REGION Network 6: CY75 interface K-reserveTakeStopperCylinder3_1
   RUNG wire#powerrail
      Contact( #AlwaysON )
      wire#w1
      Contact( #E_stop )
      wire#w2
      Coil( "ST10Cylinder".Cy[75].In.GoWorkInterlock )
   END_RUNG
   RUNG wire#w2
      Coil( "ST10Cylinder".Cy[75].In.GoHomeInterlock )
   END_RUNG
   RUNG wire#w1
      I_Contact( #AlwaysON )
      Coil( "ST10Cylinder".Cy[75].In.Error )
   END_RUNG
   // the same network as SCL:
   "ST10Cylinder".Cy[75].In.GoWorkInterlock := #AlwaysON AND #E_stop;
   "ST10Cylinder".Cy[75].In.GoHomeInterlock := #AlwaysON AND #E_stop;
   "ST10Cylinder".Cy[75].In.Error := #AlwaysON AND NOT #AlwaysON;
END_REGION

REGION Network 7: CY76 interface K-reserveTakeStopperCylinder3_2
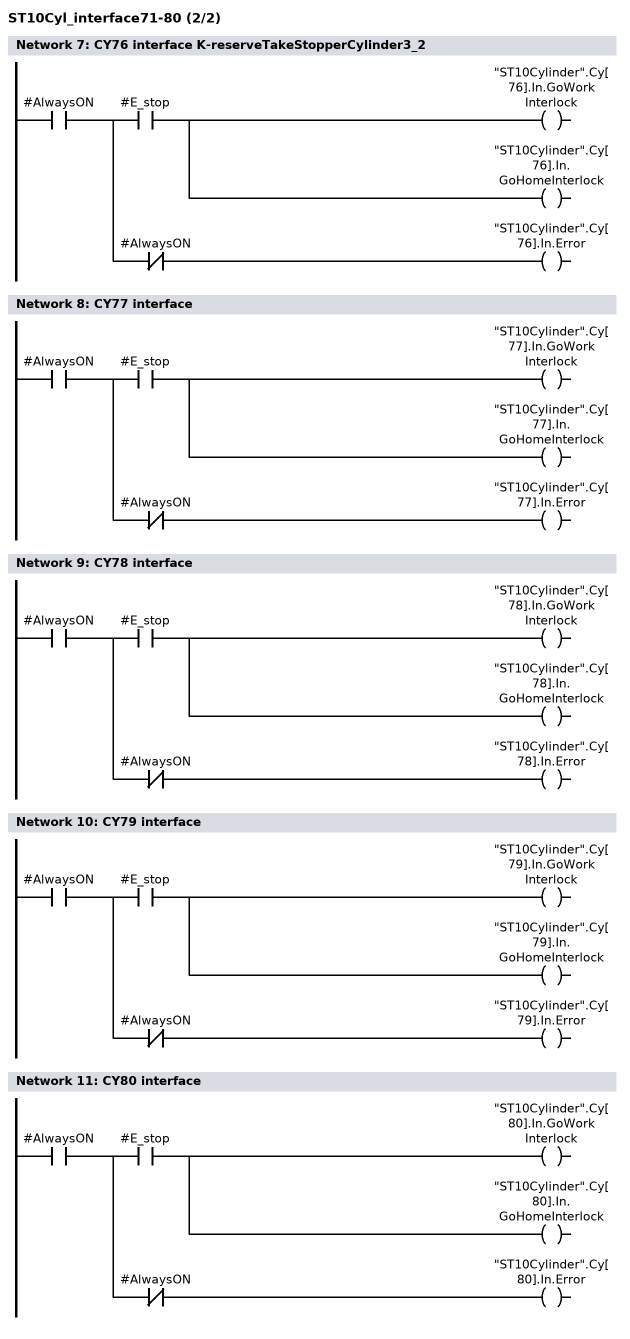
   RUNG wire#powerrail
      Contact( #AlwaysON )
      wire#w1
      Contact( #E_stop )
      wire#w2
      Coil( "ST10Cylinder".Cy[76].In.GoWorkInterlock )
   END_RUNG
   RUNG wire#w2
      Coil( "ST10Cylinder".Cy[76].In.GoHomeInterlock )
   END_RUNG
   RUNG wire#w1
      I_Contact( #AlwaysON )
      Coil( "ST10Cylinder".Cy[76].In.Error )
   END_RUNG
   // the same network as SCL:
   "ST10Cylinder".Cy[76].In.GoWorkInterlock := #AlwaysON AND #E_stop;
   "ST10Cylinder".Cy[76].In.GoHomeInterlock := #AlwaysON AND #E_stop;
   "ST10Cylinder".Cy[76].In.Error := #AlwaysON AND NOT #AlwaysON;
END_REGION

REGION Network 8: CY77 interface
   RUNG wire#powerrail
      Contact( #AlwaysON )
      wire#w1
      Contact( #E_stop )
      wire#w2
      Coil( "ST10Cylinder".Cy[77].In.GoWorkInterlock )
   END_RUNG
   RUNG wire#w2
      Coil( "ST10Cylinder".Cy[77].In.GoHomeInterlock )
   END_RUNG
   RUNG wire#w1
      I_Contact( #AlwaysON )
      Coil( "ST10Cylinder".Cy[77].In.Error )
   END_RUNG
   // the same network as SCL:
   "ST10Cylinder".Cy[77].In.GoWorkInterlock := #AlwaysON AND #E_stop;
   "ST10Cylinder".Cy[77].In.GoHomeInterlock := #AlwaysON AND #E_stop;
   "ST10Cylinder".Cy[77].In.Error := #AlwaysON AND NOT #AlwaysON;
END_REGION

REGION Network 9: CY78 interface
   RUNG wire#powerrail
      Contact( #AlwaysON )
      wire#w1
      Contact( #E_stop )
      wire#w2
      Coil( "ST10Cylinder".Cy[78].In.GoWorkInterlock )
   END_RUNG
   RUNG wire#w2
      Coil( "ST10Cylinder".Cy[78].In.GoHomeInterlock )
   END_RUNG
   RUNG wire#w1
      I_Contact( #AlwaysON )
      Coil( "ST10Cylinder".Cy[78].In.Error )
   END_RUNG
   // the same network as SCL:
   "ST10Cylinder".Cy[78].In.GoWorkInterlock := #AlwaysON AND #E_stop;
   "ST10Cylinder".Cy[78].In.GoHomeInterlock := #AlwaysON AND #E_stop;
   "ST10Cylinder".Cy[78].In.Error := #AlwaysON AND NOT #AlwaysON;
END_REGION

REGION Network 10: CY79 interface
   RUNG wire#powerrail
      Contact( #AlwaysON )
      wire#w1
      Contact( #E_stop )
      wire#w2
      Coil( "ST10Cylinder".Cy[79].In.GoWorkInterlock )
   END_RUNG
   RUNG wire#w2
      Coil( "ST10Cylinder".Cy[79].In.GoHomeInterlock )
   END_RUNG
   RUNG wire#w1
      I_Contact( #AlwaysON )
      Coil( "ST10Cylinder".Cy[79].In.Error )
   END_RUNG
   // the same network as SCL:
   "ST10Cylinder".Cy[79].In.GoWorkInterlock := #AlwaysON AND #E_stop;
   "ST10Cylinder".Cy[79].In.GoHomeInterlock := #AlwaysON AND #E_stop;
   "ST10Cylinder".Cy[79].In.Error := #AlwaysON AND NOT #AlwaysON;
END_REGION

REGION Network 11: CY80 interface
   RUNG wire#powerrail
      Contact( #AlwaysON )
      wire#w1
      Contact( #E_stop )
      wire#w2
      Coil( "ST10Cylinder".Cy[80].In.GoWorkInterlock )
   END_RUNG
   RUNG wire#w2
      Coil( "ST10Cylinder".Cy[80].In.GoHomeInterlock )
   END_RUNG
   RUNG wire#w1
      I_Contact( #AlwaysON )
      Coil( "ST10Cylinder".Cy[80].In.Error )
   END_RUNG
   // the same network as SCL:
   "ST10Cylinder".Cy[80].In.GoWorkInterlock := #AlwaysON AND #E_stop;
   "ST10Cylinder".Cy[80].In.GoHomeInterlock := #AlwaysON AND #E_stop;
   "ST10Cylinder".Cy[80].In.Error := #AlwaysON AND NOT #AlwaysON;
END_REGION
END_FUNCTION

FUNCTION "ST10Cyl_interface81-90" : Void   // FC1028, LAD
{ S7_Optimized_Access := 'FALSE' }
// stored: AutoNumber false, SetENOAutomatically false
   VAR_INPUT
      AlwaysON : Bool;
      E_stop : Bool;
   END_VAR
   VAR_TEMP
      tTest : Bool;
   END_VAR
BEGIN

REGION Network 1 (SCL): Cylinder 81-90 IO Interface (SCL)
   (*
   //Cylinder81 IO  L-UnloadingTransCylinder
   //Input
   "ST10Cylinder".Cy[81].In.WorkPositionSensor := "iL-UnloadingTransCylinderInWP";
   "ST10Cylinder".Cy[81].In.HomePositionSensor := "iL-UnloadingTransCylinderInHP";
   //Output
   "oL-UnloadingTransCylinderToWP" := "ST10Cylinder".Cy[81].Out.GoWorkPosition;
   "oL-UnloadingTransCylinderToHP" := "ST10Cylinder".Cy[81].Out.GoHomePosition;

   //Cylinder82 IO  L-UnloadingTransPalletLocationCylinder
   //Input
   "ST10Cylinder".Cy[82].In.WorkPositionSensor := "iL-UnloadingTransPalletLocationCylinderInWP";
   "ST10Cylinder".Cy[82].In.HomePositionSensor := "iL-UnloadingTransPalletLocationCylinderInHP";
   //Output
   "oL-UnloadingTransPalletLocationCylinderToWP" := "ST10Cylinder".Cy[82].Out.GoWorkPosition;
   "oL-UnloadingTransPalletLocationCylinderToHP" := "ST10Cylinder".Cy[82].Out.GoHomePosition;

   //Cylinder83 IO  L-UnloadingStopperCylinder1_1
   //Input
   "ST10Cylinder".Cy[83].In.WorkPositionSensor := "oL-UnloadingStopperCylinder1_1";
   "ST10Cylinder".Cy[83].In.HomePositionSensor := NOT "oL-UnloadingStopperCylinder1_1";
   //Output
   "oL-UnloadingStopperCylinder1_1" := "ST10Cylinder".Cy[83].Out.GoWorkPosition;
   //"oI-0030TrayLoading8trayStopperCylinderToHP" := "ST10Cylinder".Cy[83].Out.GoHomePosition;

   //Cylinder84 IO  L-UnloadingStopperCylinder1_2
   //Input
   "ST10Cylinder".Cy[84].In.WorkPositionSensor := "oL-UnloadingStopperCylinder1_2";
   "ST10Cylinder".Cy[84].In.HomePositionSensor := NOT "oL-UnloadingStopperCylinder1_2";
   //Output
   "oL-UnloadingStopperCylinder1_2" := "ST10Cylinder".Cy[84].Out.GoWorkPosition;
   //"oI-0080TrayLoadingTaketrayCylinderToHP" := "ST10Cylinder".Cy[84].Out.GoHomePosition;

   //Cylinder85 IO  L-UnloadingStopperCylinder2_1
   //Input
   "ST10Cylinder".Cy[85].In.WorkPositionSensor := "oL-UnloadingStopperCylinder2_1";
   "ST10Cylinder".Cy[85].In.HomePositionSensor := NOT "oL-UnloadingStopperCylinder2_1";
   //Output
   "oL-UnloadingStopperCylinder2_1" := "ST10Cylinder".Cy[85].Out.GoWorkPosition;
   //"oI-0050TrayLoadingTrayCylinderToHP" := "ST10Cylinder".Cy[85].Out.GoHomePosition;

   //Cylinder86  L-UnloadingStopperCylinder2_2
   //Input
   "ST10Cylinder".Cy[86].In.WorkPositionSensor := "oL-UnloadingStopperCylinder2_2";
   "ST10Cylinder".Cy[86].In.HomePositionSensor := NOT "oL-UnloadingStopperCylinder2_2";
   //Output
   "oL-UnloadingStopperCylinder2_2" := "ST10Cylinder".Cy[86].Out.GoWorkPosition;
   //"oI-0080TrayLoadingTraySupportCylinder1ToHP" := "ST10Cylinder".Cy[86].Out.GoHomePosition;

   //Cylinder87 L-UnloadingStopperCylinder3_1
   //Input
   "ST10Cylinder".Cy[87].In.WorkPositionSensor := "oL-UnloadingStopperCylinder3_1";
   "ST10Cylinder".Cy[87].In.HomePositionSensor := NOT "oL-UnloadingStopperCylinder3_1";
   //Output
   "oL-UnloadingStopperCylinder3_1" := "ST10Cylinder".Cy[87].Out.GoWorkPosition;
   //"oI-0070TrayLoadingTraySupportCylinder8ToHP" := "ST10Cylinder".Cy[87].Out.GoHomePosition;

   //Cylinder88 L-UnloadingStopperCylinder3_2
   //Input
   "ST10Cylinder".Cy[88].In.WorkPositionSensor := "oL-UnloadingStopperCylinder3_2";
   "ST10Cylinder".Cy[88].In.HomePositionSensor := NOT "oL-UnloadingStopperCylinder3_2";
   //Output
   "oL-UnloadingStopperCylinder3_2" := "ST10Cylinder".Cy[88].Out.GoWorkPosition;
   //"oI-0080TrayLoadingTrayLocationCylinderToHP" := "ST10Cylinder".Cy[88].Out.GoHomePosition;
   //
   *)
   (*
   //Cylinder89 K-reserveLoadingStopperCylinder4_1
   //Input
   "ST10Cylinder".Cy[89].In.WorkPositionSensor := "oK-reserveLoadingStopperCylinder4_1";
   "ST10Cylinder".Cy[89].In.HomePositionSensor := NOT "oK-reserveLoadingStopperCylinder4_1";
   //Output
   "oK-reserveLoadingStopperCylinder4_1" := "ST10Cylinder".Cy[89].Out.GoWorkPosition;
   //"oI-0090TrayLoadingTrayUnloadingLiftingCylinderToHP" := "ST10Cylinder".Cy[89].Out.GoHomePosition;

   //Cylinder70 K-reserveLoadingStopperCylinder4_2
   // //Input
   "ST10Cylinder".Cy[70].In.WorkPositionSensor := "oK-reserveLoadingStopperCylinder4_2";
   "ST10Cylinder".Cy[70].In.HomePositionSensor := NOT "oK-reserveLoadingStopperCylinder4_2";
   // //Output
   "oK-reserveLoadingStopperCylinder4_2" := "ST10Cylinder".Cy[70].Out.GoWorkPosition;
   // "Feeding washer  lift Cylinder ToHP" := "ST10Cylinder".Cy[70].Out.GoHomePosition;

   *)
END_REGION

REGION Network 2: CY81 interface L-UnloadingTransCylinder
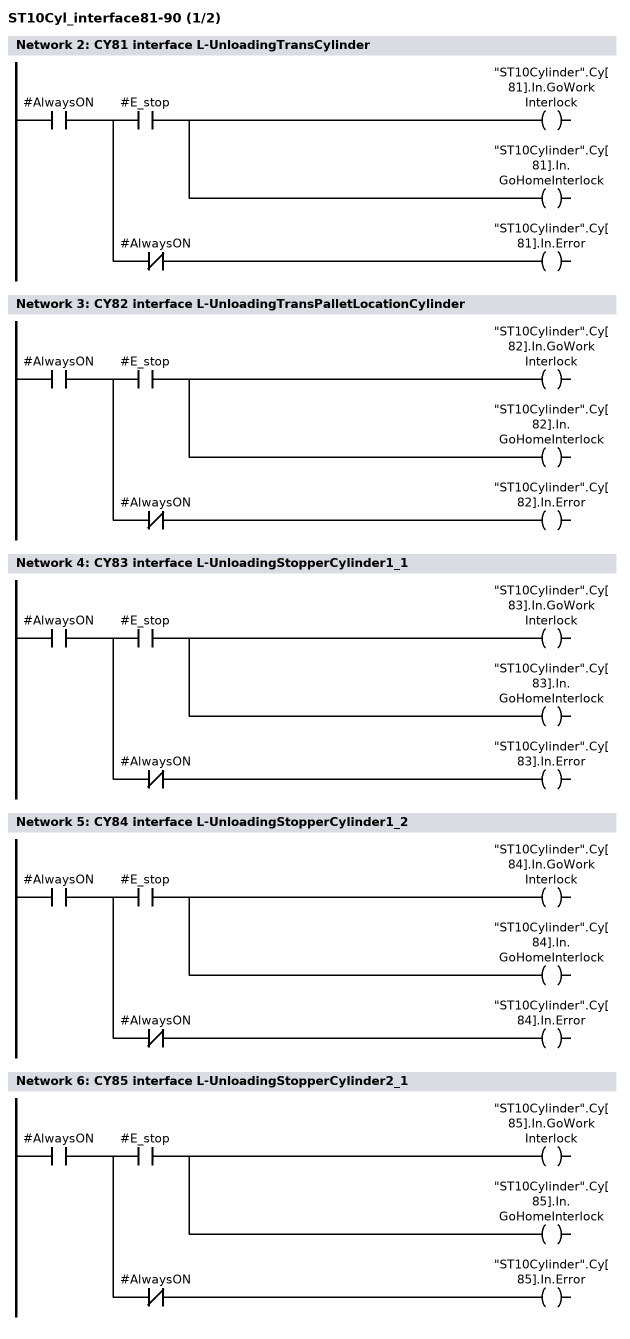
   RUNG wire#powerrail
      Contact( #AlwaysON )
      wire#w1
      Contact( #E_stop )
      wire#w2
      Coil( "ST10Cylinder".Cy[81].In.GoWorkInterlock )
   END_RUNG
   RUNG wire#w2
      Coil( "ST10Cylinder".Cy[81].In.GoHomeInterlock )
   END_RUNG
   RUNG wire#w1
      I_Contact( #AlwaysON )
      Coil( "ST10Cylinder".Cy[81].In.Error )
   END_RUNG
   // the same network as SCL:
   "ST10Cylinder".Cy[81].In.GoWorkInterlock := #AlwaysON AND #E_stop;
   "ST10Cylinder".Cy[81].In.GoHomeInterlock := #AlwaysON AND #E_stop;
   "ST10Cylinder".Cy[81].In.Error := #AlwaysON AND NOT #AlwaysON;
END_REGION

REGION Network 3: CY82 interface L-UnloadingTransPalletLocationCylinder
   RUNG wire#powerrail
      Contact( #AlwaysON )
      wire#w1
      Contact( #E_stop )
      wire#w2
      Coil( "ST10Cylinder".Cy[82].In.GoWorkInterlock )
   END_RUNG
   RUNG wire#w2
      Coil( "ST10Cylinder".Cy[82].In.GoHomeInterlock )
   END_RUNG
   RUNG wire#w1
      I_Contact( #AlwaysON )
      Coil( "ST10Cylinder".Cy[82].In.Error )
   END_RUNG
   // the same network as SCL:
   "ST10Cylinder".Cy[82].In.GoWorkInterlock := #AlwaysON AND #E_stop;
   "ST10Cylinder".Cy[82].In.GoHomeInterlock := #AlwaysON AND #E_stop;
   "ST10Cylinder".Cy[82].In.Error := #AlwaysON AND NOT #AlwaysON;
END_REGION

REGION Network 4: CY83 interface L-UnloadingStopperCylinder1_1
   RUNG wire#powerrail
      Contact( #AlwaysON )
      wire#w1
      Contact( #E_stop )
      wire#w2
      Coil( "ST10Cylinder".Cy[83].In.GoWorkInterlock )
   END_RUNG
   RUNG wire#w2
      Coil( "ST10Cylinder".Cy[83].In.GoHomeInterlock )
   END_RUNG
   RUNG wire#w1
      I_Contact( #AlwaysON )
      Coil( "ST10Cylinder".Cy[83].In.Error )
   END_RUNG
   // the same network as SCL:
   "ST10Cylinder".Cy[83].In.GoWorkInterlock := #AlwaysON AND #E_stop;
   "ST10Cylinder".Cy[83].In.GoHomeInterlock := #AlwaysON AND #E_stop;
   "ST10Cylinder".Cy[83].In.Error := #AlwaysON AND NOT #AlwaysON;
END_REGION

REGION Network 5: CY84 interface L-UnloadingStopperCylinder1_2
   RUNG wire#powerrail
      Contact( #AlwaysON )
      wire#w1
      Contact( #E_stop )
      wire#w2
      Coil( "ST10Cylinder".Cy[84].In.GoWorkInterlock )
   END_RUNG
   RUNG wire#w2
      Coil( "ST10Cylinder".Cy[84].In.GoHomeInterlock )
   END_RUNG
   RUNG wire#w1
      I_Contact( #AlwaysON )
      Coil( "ST10Cylinder".Cy[84].In.Error )
   END_RUNG
   // the same network as SCL:
   "ST10Cylinder".Cy[84].In.GoWorkInterlock := #AlwaysON AND #E_stop;
   "ST10Cylinder".Cy[84].In.GoHomeInterlock := #AlwaysON AND #E_stop;
   "ST10Cylinder".Cy[84].In.Error := #AlwaysON AND NOT #AlwaysON;
END_REGION

REGION Network 6: CY85 interface L-UnloadingStopperCylinder2_1
   RUNG wire#powerrail
      Contact( #AlwaysON )
      wire#w1
      Contact( #E_stop )
      wire#w2
      Coil( "ST10Cylinder".Cy[85].In.GoWorkInterlock )
   END_RUNG
   RUNG wire#w2
      Coil( "ST10Cylinder".Cy[85].In.GoHomeInterlock )
   END_RUNG
   RUNG wire#w1
      I_Contact( #AlwaysON )
      Coil( "ST10Cylinder".Cy[85].In.Error )
   END_RUNG
   // the same network as SCL:
   "ST10Cylinder".Cy[85].In.GoWorkInterlock := #AlwaysON AND #E_stop;
   "ST10Cylinder".Cy[85].In.GoHomeInterlock := #AlwaysON AND #E_stop;
   "ST10Cylinder".Cy[85].In.Error := #AlwaysON AND NOT #AlwaysON;
END_REGION

REGION Network 7: CY86 interface L-UnloadingStopperCylinder2_2
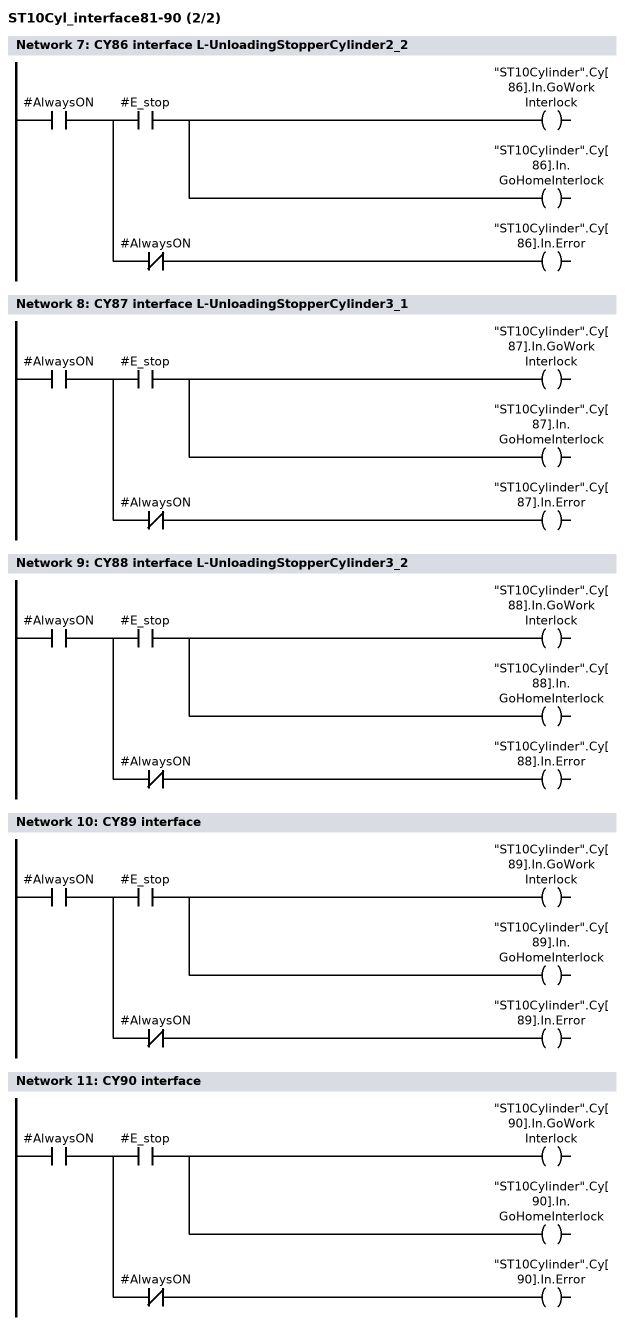
   RUNG wire#powerrail
      Contact( #AlwaysON )
      wire#w1
      Contact( #E_stop )
      wire#w2
      Coil( "ST10Cylinder".Cy[86].In.GoWorkInterlock )
   END_RUNG
   RUNG wire#w2
      Coil( "ST10Cylinder".Cy[86].In.GoHomeInterlock )
   END_RUNG
   RUNG wire#w1
      I_Contact( #AlwaysON )
      Coil( "ST10Cylinder".Cy[86].In.Error )
   END_RUNG
   // the same network as SCL:
   "ST10Cylinder".Cy[86].In.GoWorkInterlock := #AlwaysON AND #E_stop;
   "ST10Cylinder".Cy[86].In.GoHomeInterlock := #AlwaysON AND #E_stop;
   "ST10Cylinder".Cy[86].In.Error := #AlwaysON AND NOT #AlwaysON;
END_REGION

REGION Network 8: CY87 interface L-UnloadingStopperCylinder3_1
   RUNG wire#powerrail
      Contact( #AlwaysON )
      wire#w1
      Contact( #E_stop )
      wire#w2
      Coil( "ST10Cylinder".Cy[87].In.GoWorkInterlock )
   END_RUNG
   RUNG wire#w2
      Coil( "ST10Cylinder".Cy[87].In.GoHomeInterlock )
   END_RUNG
   RUNG wire#w1
      I_Contact( #AlwaysON )
      Coil( "ST10Cylinder".Cy[87].In.Error )
   END_RUNG
   // the same network as SCL:
   "ST10Cylinder".Cy[87].In.GoWorkInterlock := #AlwaysON AND #E_stop;
   "ST10Cylinder".Cy[87].In.GoHomeInterlock := #AlwaysON AND #E_stop;
   "ST10Cylinder".Cy[87].In.Error := #AlwaysON AND NOT #AlwaysON;
END_REGION

REGION Network 9: CY88 interface L-UnloadingStopperCylinder3_2
   RUNG wire#powerrail
      Contact( #AlwaysON )
      wire#w1
      Contact( #E_stop )
      wire#w2
      Coil( "ST10Cylinder".Cy[88].In.GoWorkInterlock )
   END_RUNG
   RUNG wire#w2
      Coil( "ST10Cylinder".Cy[88].In.GoHomeInterlock )
   END_RUNG
   RUNG wire#w1
      I_Contact( #AlwaysON )
      Coil( "ST10Cylinder".Cy[88].In.Error )
   END_RUNG
   // the same network as SCL:
   "ST10Cylinder".Cy[88].In.GoWorkInterlock := #AlwaysON AND #E_stop;
   "ST10Cylinder".Cy[88].In.GoHomeInterlock := #AlwaysON AND #E_stop;
   "ST10Cylinder".Cy[88].In.Error := #AlwaysON AND NOT #AlwaysON;
END_REGION

REGION Network 10: CY89 interface
   RUNG wire#powerrail
      Contact( #AlwaysON )
      wire#w1
      Contact( #E_stop )
      wire#w2
      Coil( "ST10Cylinder".Cy[89].In.GoWorkInterlock )
   END_RUNG
   RUNG wire#w2
      Coil( "ST10Cylinder".Cy[89].In.GoHomeInterlock )
   END_RUNG
   RUNG wire#w1
      I_Contact( #AlwaysON )
      Coil( "ST10Cylinder".Cy[89].In.Error )
   END_RUNG
   // the same network as SCL:
   "ST10Cylinder".Cy[89].In.GoWorkInterlock := #AlwaysON AND #E_stop;
   "ST10Cylinder".Cy[89].In.GoHomeInterlock := #AlwaysON AND #E_stop;
   "ST10Cylinder".Cy[89].In.Error := #AlwaysON AND NOT #AlwaysON;
END_REGION

REGION Network 11: CY90 interface
   RUNG wire#powerrail
      Contact( #AlwaysON )
      wire#w1
      Contact( #E_stop )
      wire#w2
      Coil( "ST10Cylinder".Cy[90].In.GoWorkInterlock )
   END_RUNG
   RUNG wire#w2
      Coil( "ST10Cylinder".Cy[90].In.GoHomeInterlock )
   END_RUNG
   RUNG wire#w1
      I_Contact( #AlwaysON )
      Coil( "ST10Cylinder".Cy[90].In.Error )
   END_RUNG
   // the same network as SCL:
   "ST10Cylinder".Cy[90].In.GoWorkInterlock := #AlwaysON AND #E_stop;
   "ST10Cylinder".Cy[90].In.GoHomeInterlock := #AlwaysON AND #E_stop;
   "ST10Cylinder".Cy[90].In.Error := #AlwaysON AND NOT #AlwaysON;
END_REGION
END_FUNCTION

FUNCTION "ST10_ChangeOver" : Void   // FC1008, LAD
{ S7_Optimized_Access := 'FALSE' }
// stored: AutoNumber false, SetENOAutomatically false
   VAR_TEMP
      sString : String[50];
      FixtureNumber : Int;
      FixtureIndex : Int;
      tRET_VAL : Int;
   END_VAR
BEGIN

REGION Network 1: Recipe Active
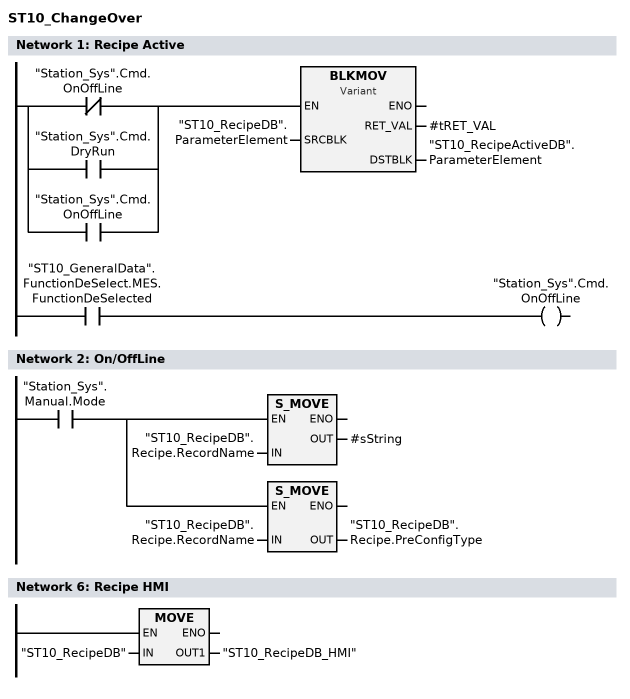
   RUNG wire#powerrail
      I_Contact( "Station_Sys".Cmd.OnOffLine )
      wire#w1
      { S7_Templates := "blk_type := Variant" } BLKMOV(SRCBLK := "ST10_RecipeDB".ParameterElement, RET_VAL => #tRET_VAL, DSTBLK => "ST10_RecipeActiveDB".ParameterElement)
   END_RUNG
   RUNG wire#powerrail
      Contact( "Station_Sys".Cmd.DryRun )
   END_RUNG wire#w1
   RUNG wire#powerrail
      Contact( "Station_Sys".Cmd.OnOffLine )
   END_RUNG wire#w1
   RUNG wire#powerrail
      Contact( "ST10_GeneralData".FunctionDeSelect.MES.FunctionDeSelected )
      Coil( "Station_Sys".Cmd.OnOffLine )
   END_RUNG
   // the same network as SCL:
   IF NOT "Station_Sys".Cmd.OnOffLine OR "Station_Sys".Cmd.DryRun OR "Station_Sys".Cmd.OnOffLine THEN
       #tRET_VAL := BLKMOV(SRCBLK := "ST10_RecipeDB".ParameterElement,
                           DSTBLK => "ST10_RecipeActiveDB".ParameterElement);
   END_IF;
   "Station_Sys".Cmd.OnOffLine := "ST10_GeneralData".FunctionDeSelect.MES.FunctionDeSelected;
END_REGION

REGION Network 2: On/OffLine
   RUNG wire#powerrail
      Contact( "Station_Sys".Manual.Mode )
      wire#w1
      S_Move(in := "ST10_RecipeDB".Recipe.RecordName, out => #sString)
   END_RUNG
   RUNG wire#w1
      S_Move(in := "ST10_RecipeDB".Recipe.RecordName, out => "ST10_RecipeDB".Recipe.PreConfigType)
   END_RUNG
   // the same network as SCL:
   IF "Station_Sys".Manual.Mode THEN
       #sString := "ST10_RecipeDB".Recipe.RecordName;
       "ST10_RecipeDB".Recipe.PreConfigType := "ST10_RecipeDB".Recipe.RecordName;
   END_IF;
END_REGION

NETWORK
TITLE = 换型功能块调用 / Transposition function block call
//"ST10_RecipeDB".Recipe.PreConfigType    AUTO CONFIG, When PLC activate change over, Set Recipe data record Tags
//"ST10_RecipeDB".ParameterElement.TypeName    HMI MANUAL CONFIG, HMI Recipe data record element:Product_type
//HMI Recipe data record element Product_type set value must be same with HMI Recipe data record Name

      A     "ChangeOver_DB".Global.ChangeOverActive;
      A     "Station_Sys".Auto.Mode;
      =     "ST10_RecipeDB".Recipe.Trigger;

      CALL  "ChangeOver"
      ( iCheckType      := "ST10_RecipeDB".ParameterElement.TypeName,
        "iPulse*500ms"  := "Sys".COM.FlashTime500mS,
        iReset          := "Station_Sys".Cmd.Reset,
        Ret_Val         := "ST10_RecipeDB".Recipe.Ret,
        oPulse          := "ST10_RecipeDB".Recipe.Pulse,
        oEqual          := "ST10_RecipeDB".Recipe.Equal,  // CheckType=PreConfigType, indicate ChangerOver successfully
        ioPreConfigType := "ST10_RecipeDB".Recipe.PreConfigType,
        ioCurrentName   := "ST10_RecipeDB".Recipe.RecordName,
        iotime          := "ST10_RecipeDB".Recipe."time",
        ioTrigger       := "ST10_RecipeDB".Recipe.Trigger,
        ioPosEdg        := "ST10_RecipeDB".Recipe.PosEdg,
        ioAlarm         := "ST10_RecipeDB".Recipe.Alarm,
        ioPls           := "ST10_RecipeDB".Recipe.Pls
      );




REGION Network 4 (SCL): Fixture换型工装 / Fixture Changing fixture
   //Fixture 1 输入轴换型X轴工装
   //工装检测屏蔽条件
   "ST10_GeneralData".FixtureIDCheck[1].FixtureCheckUnEnable := 0;

   //工装检测传感器赋值

   "ST10_GeneralData".FixtureIDCheck[1].FixtureIDCheckValue.%X0 := 0;
   "ST10_GeneralData".FixtureIDCheck[1].FixtureIDCheckValue.%X1 := 0;
   "ST10_GeneralData".FixtureIDCheck[1].FixtureIDCheckValue.%X2 := 0;
   "ST10_GeneralData".FixtureIDCheck[1].FixtureIDCheckValue.%X3 := 0;
   "ST10_GeneralData".FixtureIDCheck[1].FixtureIDCheckValue.%X4 := 0;
   "ST10_GeneralData".FixtureIDCheck[1].FixtureIDCheckValue.%X5 := 0;
   "ST10_GeneralData".FixtureIDCheck[1].FixtureIDCheckValue.%X6 := 0;
   "ST10_GeneralData".FixtureIDCheck[1].FixtureIDCheckValue.%X7 := 0;
END_REGION

REGION Network 5 (SCL): FixtureID Check Call
   //循环数量为工装检测的数量

   #FixtureNumber := 1;

   //工装检测功能块调用

   #FixtureIndex := 1;

   FOR #FixtureIndex := 1 TO #FixtureNumber DO

       "fcFixtureCheck"(iRecipeSetValue := "ST10_RecipeDB".ParameterElement.FixtureID[#FixtureIndex],
                        FixtureIDCheck := "ST10_GeneralData".FixtureIDCheck[#FixtureIndex]);

   END_FOR;
END_REGION

REGION Network 6: Recipe HMI
   RUNG wire#powerrail
      Move(in := "ST10_RecipeDB", out1 => "ST10_RecipeDB_HMI")
   END_RUNG
   // the same network as SCL:
   "ST10_RecipeDB_HMI" := "ST10_RecipeDB";
END_REGION
END_FUNCTION

FUNCTION "ChangeOver" : Bool   // FC3002, SCL
TITLE = ChangeOverV3
{ S7_Optimized_Access := 'FALSE' }
AUTHOR : STD
FAMILY : RCS
VERSION : 18.0
// stored: AutoNumber false, SetENOAutomatically true
   VAR_INPUT
      iCheckType : String;   // Person Confirm input type ID/NAME
      "iPulse*500ms" : Bool;   // pulse
      iReset : Bool;
   END_VAR
   VAR_OUTPUT
      oPulse : Bool;   // system pulse[HMI Variable Must keep continous mode]
      oEqual : Bool;
   END_VAR
   VAR_IN_OUT
      ioPreConfigType : String;   // to be changed recipe ID/NAME
      ioCurrentName : String;   // current recipe record name
      iotime : Int;   // time record
      ioTrigger : Bool;   // trigger for changeing over
      ioPosEdg : Bool;   // postive edge bit
      ioAlarm : Bool;   // Changover time out
      ioPls : Bool;
   END_VAR
   VAR_TEMP
      tpPosEdg : Bool;
      tpPls : Bool;
   END_VAR
   // Ret_Val : 0-NG/1-OK
BEGIN
   //---------------------------------------------------------------//
   //FunctionName:ChangeOverV3
   //FunctionDescription:ChangeOver
   //---------------------------------------------------------------//
   (*in:

   iPreConfigType  String
   iLastType   String
   iPulse*500ms    Bool
   iTrigger    Bool


   //inout:
   //out:
   oPulse  Bool
   oAlarm  Bool

   *)
   //---------------------------------------------------------------//
   //Version:V2
   //D&T:2016-11-125
   //Group:RCS
   //Author:JM
   //-------------------------Modify1----------------------------------//
   //Version:V3.0
   //D&T:2016-11-28
   //Group: RCS
   //Author:JM
   //Modify: add timeout bit 
   //-------------------------Modify2----------------------------------//
   //Version:V3.0
   //D&T:20180416
   //Group: RCS
   //Author:JM
   //Modify:
   // Add pls flag in order to keep paramter that download after modifier safe.
   #tpPls := #ioTrigger AND NOT #ioPls;
   #ioPls := #ioTrigger;
   #tpPosEdg := #"iPulse*500ms" AND NOT #ioPosEdg;
   #ioPosEdg := #"iPulse*500ms";
   #oEqual := #ioPreConfigType = #iCheckType AND #ioPreConfigType<>'';


   // IF #tpPls THEN
   //     #ioPreConfigType:='';
   // END_IF;
   IF (#iReset AND #ioAlarm) OR #oEqual THEN
       #ioAlarm := 0;
   END_IF;
   IF NOT #ioTrigger THEN
       #ChangeOver := 0;
       #iotime := 0;
       // #oAlarm := 0;
       RETURN;
   ELSE
       IF #tpPosEdg THEN
           #iotime := #iotime + 1;
       END_IF;
       IF #iotime >= 10 THEN
           #ioAlarm := 1;
           #ioTrigger := 0;
           // ELSE
           //     #oAlarm := 0;
       END_IF;
       #ChangeOver := 0;
       // #tpCurrentProductlen := LEN(#tpCurrentProduct);
       // #tpLastProductlen := LEN(#tpLastProduct);
       IF #ioPreConfigType <> #iCheckType THEN
           #oPulse := #"iPulse*500ms";
           RETURN;
       ELSE
           IF #ioCurrentName <> #ioPreConfigType THEN
               #ioCurrentName := #ioPreConfigType;
           END_IF;
           #iotime := 0;
           #ioAlarm := 0;
           #oPulse := 0;
           #ChangeOver := 1;
           #ioTrigger := 0;
           ENO := 1;
       END_IF;

   END_IF;
END_FUNCTION

FUNCTION "ST10_Device" : Void   // FC1010, LAD
{ S7_Optimized_Access := 'TRUE' }
// stored: AutoNumber false, SetENOAutomatically false
   VAR_INPUT
      iSysMode : "RCS_SysComInterface_V1";
   END_VAR
BEGIN

NETWORK
TITLE = SafetyGate

      CALL  "ST10_SafetyGate"
      ( iSysMode := #iSysMode
      );


NETWORK
TITLE = PartData

      CALL  "ST10_PartData"
      ( iSysMode := #iSysMode
      );


NETWORK
TITLE = Analog

      CALL  "ST10_Analog"
      ( iSysMode := #iSysMode
      );


REGION Network 4: SR Scan
END_REGION

REGION Network 7: CuringOven
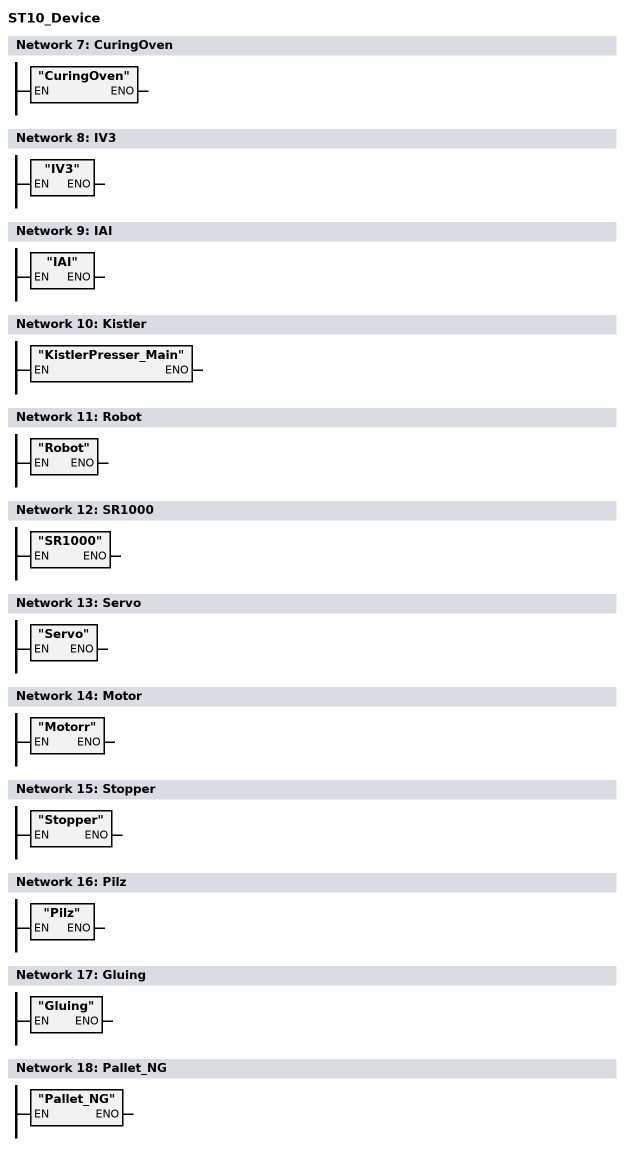
   RUNG wire#powerrail
      "CuringOven"()
   END_RUNG
   // the same network as SCL:
   "CuringOven"();
END_REGION

REGION Network 8: IV3
   RUNG wire#powerrail
      "IV3"()
   END_RUNG
   // the same network as SCL:
   "IV3"();
END_REGION

REGION Network 9: IAI
   RUNG wire#powerrail
      "IAI"()
   END_RUNG
   // the same network as SCL:
   "IAI"();
END_REGION

REGION Network 10: Kistler
   RUNG wire#powerrail
      "KistlerPresser_Main"()
   END_RUNG
   // the same network as SCL:
   "KistlerPresser_Main"();
END_REGION

REGION Network 11: Robot
   RUNG wire#powerrail
      "Robot"()
   END_RUNG
   // the same network as SCL:
   "Robot"();
END_REGION

REGION Network 12: SR1000
   RUNG wire#powerrail
      "SR1000"()
   END_RUNG
   // the same network as SCL:
   "SR1000"();
END_REGION

REGION Network 13: Servo
   RUNG wire#powerrail
      "Servo"()
   END_RUNG
   // the same network as SCL:
   "Servo"();
END_REGION

REGION Network 14: Motor
   RUNG wire#powerrail
      "Motorr"()
   END_RUNG
   // the same network as SCL:
   "Motorr"();
END_REGION

REGION Network 15: Stopper
   RUNG wire#powerrail
      "Stopper"()
   END_RUNG
   // the same network as SCL:
   "Stopper"();
END_REGION

REGION Network 16: Pilz
   RUNG wire#powerrail
      "Pilz"()
   END_RUNG
   // the same network as SCL:
   "Pilz"();
END_REGION

REGION Network 17: Gluing
   RUNG wire#powerrail
      "Gluing"()
   END_RUNG
   // the same network as SCL:
   "Gluing"();
END_REGION

REGION Network 18: Pallet_NG
   RUNG wire#powerrail
      "Pallet_NG"()
   END_RUNG
   // the same network as SCL:
   "Pallet_NG"();
END_REGION
END_FUNCTION

FUNCTION "ST10_SafetyGate" : Void   // FC1140, SCL
{ S7_Optimized_Access := 'TRUE' }
// stored: AutoNumber false, SetENOAutomatically false
   VAR_INPUT
      iSysMode : "RCS_SysComInterface_V1";
   END_VAR
   VAR_TEMP
      idex : Int;
   END_VAR
BEGIN


   REGION SafetyGate 1    
       //定义编号
       #idex := 1;
       //功能块调用
       //
       "ST10_SafetyGate1_DB"(iSysInface := #iSysMode,
                             "iSafetyGate Opened Monitor" := NOT "iSafety door Locking FeedBack_1",
                             "iSafetyGate Locked Monitor" := "ST10_SysOutput".SafetyDoorCoil[1],
                             i1s_Pulse := "ClockMemory1s",
                             iMode :=1,
                              "oSafetyGate LockedLamp"=>"ST10_SafetyGate_InterfaceDB" .SafetyDoorLamp[1],
                              ioSafetyGateLock := "ST10_SysOutput".SafetyDoorCoil[1],
                              ioHMI_Interface := "ST10_SafetyGate_InterfaceDB".aDev[#idex]);

   END_REGION

   REGION SafetyGate 2    
       //定义编号
       #idex := 2;
       //功能块调用
       //
       "ST10_SafetyGate2_DB"(iSysInface := #iSysMode,
                             "iSafetyGate Opened Monitor" := NOT "iSafety door Locking FeedBack_2",
                             "iSafetyGate Locked Monitor" := "ST10_SysOutput".SafetyDoorCoil[2],
                             i1s_Pulse := "ClockMemory1s",
                             iMode :=1,
                              "oSafetyGate LockedLamp"=> "ST10_SafetyGate_InterfaceDB" .SafetyDoorLamp[2],
                              ioSafetyGateLock := "ST10_SysOutput".SafetyDoorCoil[2],
                              ioHMI_Interface := "ST10_SafetyGate_InterfaceDB".aDev[#idex]);

   END_REGION

   REGION SafetyGate 3    
       //定义编号
       #idex := 3;
       //功能块调用
       //
       "ST10_SafetyGate3_DB"(iSysInface := #iSysMode,
                             "iSafetyGate Opened Monitor" := NOT "iSafety door Locking FeedBack_3",
                             "iSafetyGate Locked Monitor" := "ST10_SysOutput".SafetyDoorCoil[3],
                             i1s_Pulse := "ClockMemory1s",
                             iMode :=1,
                              "oSafetyGate LockedLamp"=> "ST10_SafetyGate_InterfaceDB" .SafetyDoorLamp[3],
                              ioSafetyGateLock := "ST10_SysOutput".SafetyDoorCoil[3],
                              ioHMI_Interface := "ST10_SafetyGate_InterfaceDB".aDev[#idex]);

   END_REGION

   REGION SafetyGate 4    
       //定义编号
       #idex := 4;
       //功能块调用
       //
       "ST10_SafetyGate4_DB"(iSysInface := #iSysMode,
                              "iSafetyGate Opened Monitor" := NOT "iSafety door Locking FeedBack_4",
                              "iSafetyGate Locked Monitor" := "ST10_SysOutput".SafetyDoorCoil[4],
                              i1s_Pulse := "ClockMemory1s",
                              iMode :=1,
                              "oSafetyGate LockedLamp"=>"ST10_SafetyGate_InterfaceDB" .SafetyDoorLamp[4],
                              ioSafetyGateLock := "ST10_SysOutput".SafetyDoorCoil[4],
                              ioHMI_Interface := "ST10_SafetyGate_InterfaceDB".aDev[#idex]);

   END_REGION

   REGION SafetyGate 5    
       //定义编号
       #idex := 5;
       //功能块调用
       //
       "ST10_SafetyGate5_DB"(iSysInface := #iSysMode,
                             "iSafetyGate Opened Monitor" := NOT "iSafety door Locking FeedBack_5",
                             "iSafetyGate Locked Monitor" := "ST10_SysOutput".SafetyDoorCoil[5],
                             i1s_Pulse := "ClockMemory1s",
                             iMode :=1,
                             "oSafetyGate LockedLamp" => "ST10_SafetyGate_InterfaceDB".SafetyDoorLamp[5],
                             ioSafetyGateLock := "ST10_SysOutput".SafetyDoorCoil[5],
                             ioHMI_Interface := "ST10_SafetyGate_InterfaceDB".aDev[#idex]);

   END_REGION

   REGION SafetyGate 6    
       //定义编号
       #idex := 6;
       //功能块调用
       //
       "ST10_SafetyGate6_DB"(iSysInface := #iSysMode,
                             "iSafetyGate Opened Monitor" := NOT "iSafety door Locking FeedBack_6",
                             "iSafetyGate Locked Monitor" := "ST10_SysOutput".SafetyDoorCoil[6],
                             i1s_Pulse := "ClockMemory1s",
                             iMode :=1,
                             "oSafetyGate LockedLamp" => "ST10_SafetyGate_InterfaceDB".SafetyDoorLamp[6],
                             ioSafetyGateLock := "ST10_SysOutput".SafetyDoorCoil[6],
                             ioHMI_Interface := "ST10_SafetyGate_InterfaceDB".aDev[#idex]);

                          END_REGION

   REGION SafetyGate 7    
       //定义编号
       #idex := 7;
       //功能块调用
       //
       "ST10_SafetyGate7_DB"(iSysInface := #iSysMode,
                             "iSafetyGate Opened Monitor" := NOT "iSafety door Locking FeedBack_7",
                             "iSafetyGate Locked Monitor" := "ST10_SysOutput".SafetyDoorCoil[7],
                             i1s_Pulse := "ClockMemory1s",
                             iMode :=1,
                             "oSafetyGate LockedLamp" => "ST10_SafetyGate_InterfaceDB".SafetyDoorLamp[7],
                             ioSafetyGateLock := "ST10_SysOutput".SafetyDoorCoil[7],
                             ioHMI_Interface := "ST10_SafetyGate_InterfaceDB".aDev[#idex]);

   END_REGION

   REGION SafetyGate 8    
       //定义编号
       #idex := 8;
       //功能块调用
       //
       "ST10_SafetyGate8_DB"(iSysInface := #iSysMode,
                             "iSafetyGate Opened Monitor" := NOT "iSafety door Locking FeedBack_8",
                             "iSafetyGate Locked Monitor" := "ST10_SysOutput".SafetyDoorCoil[8],
                             i1s_Pulse := "ClockMemory1s",
                             iMode :=1,
                             "oSafetyGate LockedLamp" => "ST10_SafetyGate_InterfaceDB".SafetyDoorLamp[8],
                             ioSafetyGateLock := "ST10_SysOutput".SafetyDoorCoil[8],
                             ioHMI_Interface := "ST10_SafetyGate_InterfaceDB".aDev[#idex]);

                          END_REGION

   REGION SafetyGate 9    
    //定义编号
     #idex := 9;
    //功能块调用
    //
      "ST10_SafetyGate9_DB"(iSysInface := #iSysMode,
                            "iSafetyGate Opened Monitor" := NOT "iSafety Door Locking FeedBack",
                           "iSafetyGate Locked Monitor" := "ST10_SysOutput".SafetyDoorCoil[9],
                           i1s_Pulse := "ClockMemory1s",
                           iMode :=1,
                            "oSafetyGate LockedLamp" => "ST10_SafetyGate_InterfaceDB".SafetyDoorLamp[9],
                            ioSafetyGateLock := "ST10_SysOutput".SafetyDoorCoil[9],
                            ioHMI_Interface := "ST10_SafetyGate_InterfaceDB".aDev[#idex]);

   END_REGION

   REGION SafetyGate 11    
    //定义编号
   #idex := 11;
   //功能块调用
   //
   "ST10_MaterialGate1_DB"(iSysInface := #iSysMode,
                           "iSafetyGate Opened Monitor" := NOT "iMateriel Door Locking FeedBack_H1",
                          "iSafetyGate Locked Monitor" := "ST10_SysOutput".MaterialDoorCoil[1],
                          i1s_Pulse := "ClockMemory1s",
                          iMode :=2,
                            "oSafetyGate LockedLamp" => "ST10_SafetyGate_InterfaceDB".SafetyDoorLamp[11],
                            ioSafetyGateLock := "ST10_SysOutput".MaterialDoorCoil[1],
                            ioHMI_Interface := "ST10_SafetyGate_InterfaceDB".aDev[#idex]);

   END_REGION

   REGION SafetyGate 12    
       //定义编号
       #idex := 12;
       //功能块调用
       //
       "ST10_MaterialGate2_DB"(iSysInface := #iSysMode,
                               "iSafetyGate Opened Monitor" := NOT "iMateriel Door Locking FeedBack_H2",
                             "iSafetyGate Locked Monitor" := "ST10_SysOutput".MaterialDoorCoil[2],
                             i1s_Pulse := "ClockMemory1s",
                             iMode :=2,
                             "oSafetyGate LockedLamp" => "ST10_SafetyGate_InterfaceDB".SafetyDoorLamp[12],
                             ioSafetyGateLock := "ST10_SysOutput".MaterialDoorCoil[2],
                             ioHMI_Interface := "ST10_SafetyGate_InterfaceDB".aDev[#idex]);

   END_REGION

   REGION SafetyGate 13    
       //定义编号
       #idex := 13;
       //功能块调用
       //
       "ST10_MaterialGate3_DB"(iSysInface := #iSysMode,
                               "iSafetyGate Opened Monitor" := NOT "iMateriel Door Locking FeedBack_J1",
                             "iSafetyGate Locked Monitor" := "ST10_SysOutput".MaterialDoorCoil[3],
                             i1s_Pulse := "ClockMemory1s",
                             iMode :=2,
                             "oSafetyGate LockedLamp" => "ST10_SafetyGate_InterfaceDB".SafetyDoorLamp[13],
                             ioSafetyGateLock := "ST10_SysOutput".MaterialDoorCoil[3],
                             ioHMI_Interface := "ST10_SafetyGate_InterfaceDB".aDev[#idex]);

   END_REGION

   REGION SafetyGate 14    
       //定义编号
       #idex := 14;
       //功能块调用
       //
       "ST10_MaterialGate4_DB"(iSysInface := #iSysMode,
                               "iSafetyGate Opened Monitor" := NOT "iMateriel Door Locking FeedBack_J2",
                             "iSafetyGate Locked Monitor" := "ST10_SysOutput".MaterialDoorCoil[4],
                             i1s_Pulse := "ClockMemory1s",
                             iMode :=2,
                             "oSafetyGate LockedLamp" => "ST10_SafetyGate_InterfaceDB".SafetyDoorLamp[14],
                             ioSafetyGateLock := "ST10_SysOutput".MaterialDoorCoil[4],
                             ioHMI_Interface := "ST10_SafetyGate_InterfaceDB".aDev[#idex]);

   END_REGION

   REGION SafetyGate 15    
       //定义编号
       #idex := 15;
       //功能块调用
       //
       "ST10_MaterialGate5_DB"(iSysInface := #iSysMode,
                               "iSafetyGate Opened Monitor" := NOT "iMateriel Door Locking FeedBack_K1",
                             "iSafetyGate Locked Monitor" := "ST10_SysOutput".MaterialDoorCoil[5],
                             i1s_Pulse := "ClockMemory1s",
                             iMode :=2,
                             "oSafetyGate LockedLamp" => "ST10_SafetyGate_InterfaceDB".SafetyDoorLamp[15],
                             ioSafetyGateLock := "ST10_SysOutput".MaterialDoorCoil[5],
                             ioHMI_Interface := "ST10_SafetyGate_InterfaceDB".aDev[#idex]);

   END_REGION

   REGION SafetyGate 16    
       //定义编号
       #idex := 16;
       //功能块调用
       //
       "ST10_MaterialGate6_DB"(iSysInface := #iSysMode,
                               "iSafetyGate Opened Monitor" := NOT "iMateriel Door Locking FeedBack_K2",
                               "iSafetyGate Locked Monitor" := "ST10_SysOutput".MaterialDoorCoil[6],
                               i1s_Pulse := "ClockMemory1s",
                               iMode :=2,
                               "oSafetyGate LockedLamp" => "ST10_SafetyGate_InterfaceDB".SafetyDoorLamp[16],
                               ioSafetyGateLock := "ST10_SysOutput".MaterialDoorCoil[6],
                               ioHMI_Interface := "ST10_SafetyGate_InterfaceDB".aDev[#idex]);

   END_REGION

   REGION SafetyGate 17    
       //定义编号
       #idex := 17;
       //功能块调用
       //
       "ST10_MaterialGate7_DB"(iSysInface := #iSysMode,
                               "iSafetyGate Opened Monitor" := NOT "iMateriel Door Locking FeedBack_L1",
                               "iSafetyGate Locked Monitor" := "ST10_SysOutput".MaterialDoorCoil[7],
                               i1s_Pulse := "ClockMemory1s",
                               iMode :=2,
                             "oSafetyGate LockedLamp" => "ST10_SafetyGate_InterfaceDB".SafetyDoorLamp[17],
                             ioSafetyGateLock := "ST10_SysOutput".MaterialDoorCoil[7],
                             ioHMI_Interface := "ST10_SafetyGate_InterfaceDB".aDev[#idex]);

   END_REGION

   REGION SafetyGate 18    
       //定义编号
       #idex := 18;
       //功能块调用
       //
       "ST10_NGGate1_DB"(iSysInface := #iSysMode,
                         "iSafetyGate Opened Monitor" :=  "iE-NG-01 Safety Gate_Open",
                         "iSafetyGate Locked Monitor" := "iE-NG-01 Safety Gate_UnLock",
                               i1s_Pulse := "ClockMemory1s",
                               iMode := 2,
                               "oSafetyGate LockedLamp" => "ST10_SafetyGate_InterfaceDB".SafetyDoorLamp[18],
                               ioSafetyGateLock := "ST10_SysOutput".MaterialDoorCoil[8],
                               ioHMI_Interface := "ST10_SafetyGate_InterfaceDB".aDev[#idex]);

   END_REGION

   REGION SafetyGate 19    
       //定义编号
       #idex := 19;
       //功能块调用
       //
       "ST10_NGGate2_DB"(iSysInface := #iSysMode,
                         "iSafetyGate Opened Monitor" := "iE-NG-02 Safety Gate_Open",
                         "iSafetyGate Locked Monitor" := "iE-NG-02 Safety Gate_UnLock",
                         i1s_Pulse := "ClockMemory1s",
                         iMode := 2,
                         "oSafetyGate LockedLamp" => "ST10_SafetyGate_InterfaceDB".SafetyDoorLamp[19],
                         ioSafetyGateLock := "ST10_SysOutput".MaterialDoorCoil[9],
                         ioHMI_Interface := "ST10_SafetyGate_InterfaceDB".aDev[#idex]);

   END_REGION
END_FUNCTION

FUNCTION_BLOCK "SafetyGate"   // FB5200, LAD
{ S7_Optimized_Access := 'FALSE' }
// stored: AutoNumber false, SetENOAutomatically false
   VAR_INPUT
      iSysInface : "RCS_SysComInterface_V1";
      "iSafetyGate Opened Monitor" : Bool;   // 安全门打开状态监控
      "iSafetyGate Locked Monitor" : Bool;   // 安全门锁定状态监控
      i1s_Pulse : Bool;   // 1s脉冲信号
      "iSafetyGate AutoLock Timer" : Time := T#1s;   // 安全门自动模式下锁延时
      "iSafetyGate ManualLock Timer" : Time := T#60s;   // 安全门手动模式下锁定延时
      iMode : Int;
   END_VAR
   VAR_OUTPUT
      "oSafetyGate LockedLamp" { ExternalAccessible := 'False'; ExternalVisible := 'False'; ExternalWritable := 'False'} : Bool;   // 安全门解锁输出状态
   END_VAR
   VAR_IN_OUT
      ioSafetyGateLock : Bool;   // 安全门锁定输出
      ioHMI_Interface : "SafetyGateUDT";
   END_VAR
   VAR
      "sSafetyGate Timer" { S7_SetPoint := 'True'} : Array[1..5] of TON_TIME;
      sP_Trig : Array[1..10] of Bool;
      sN_Trig : Array[1..10] of Bool;
      "sSafetyGate UnlockRequest" { ExternalAccessible := 'False'; ExternalVisible := 'False'; ExternalWritable := 'False'} : Bool;   // 安全门开门请求标志位
      "sSafetyGate LockRequest" : Bool;
   END_VAR
   VAR_TEMP
      tAlyways_On : Bool;
      tAlyways_Off : Bool;
   END_VAR
   VAR_TEMP   // added for the SCL form of the ladder/FBD networks
      _w1 : Bool;
      _w2 : Bool;
      _w3 : Bool;
      _w4 : Bool;
      _w5 : Bool;
   END_VAR
BEGIN

REGION Network 1: #tAlyways_On
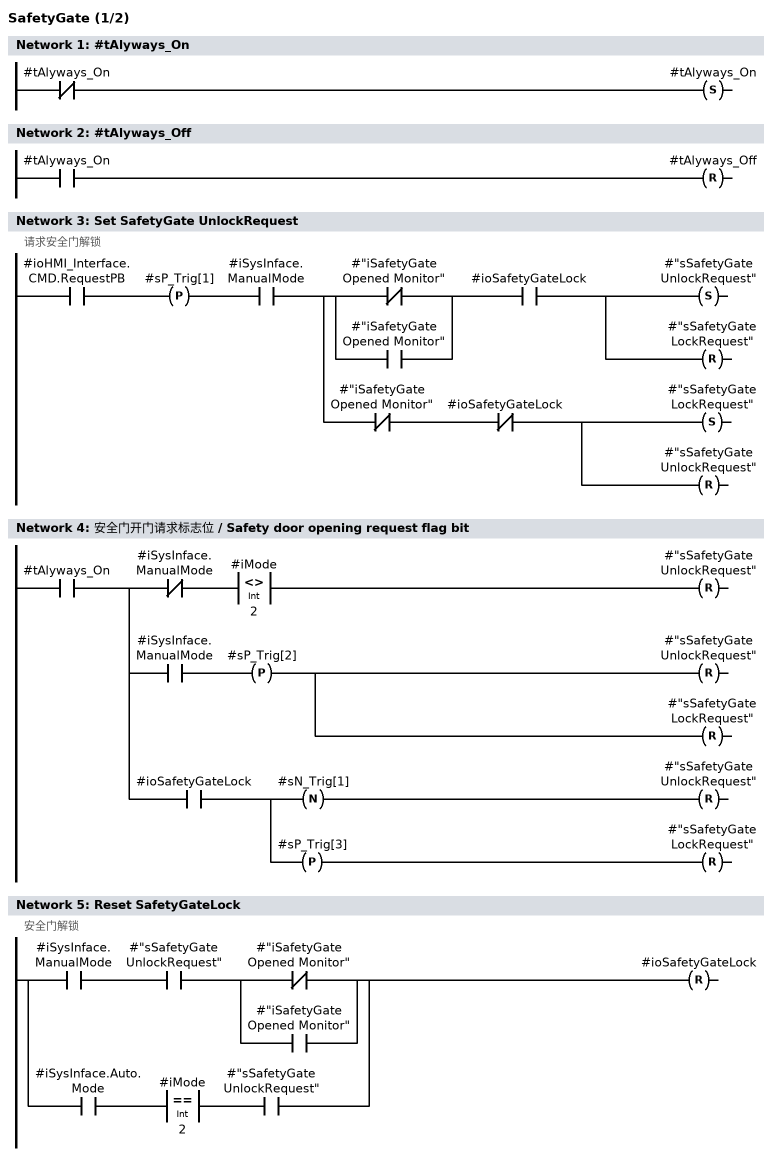
   RUNG wire#powerrail
      I_Contact( #tAlyways_On )
      S_Coil( #tAlyways_On )
   END_RUNG
   // the same network as SCL:
   IF NOT #tAlyways_On THEN #tAlyways_On := TRUE; END_IF;
END_REGION

REGION Network 2: #tAlyways_Off
   RUNG wire#powerrail
      Contact( #tAlyways_On )
      R_Coil( #tAlyways_Off )
   END_RUNG
   // the same network as SCL:
   IF #tAlyways_On THEN #tAlyways_Off := FALSE; END_IF;
END_REGION

REGION Network 3: Set SafetyGate UnlockRequest
   // 请求安全门解锁
   RUNG wire#powerrail
      Contact( #ioHMI_Interface.CMD.RequestPB )
      P_Trig( #sP_Trig[1] )
      Contact( #iSysInface.ManualMode )
      wire#w1
      I_Contact( #"iSafetyGate Opened Monitor" )
      wire#w2
      Contact( #ioSafetyGateLock )
      wire#w3
      S_Coil( #"sSafetyGate UnlockRequest" )
   END_RUNG
   RUNG wire#w1
      Contact( #"iSafetyGate Opened Monitor" )
   END_RUNG wire#w2
   RUNG wire#w3
      R_Coil( #"sSafetyGate LockRequest" )
   END_RUNG
   RUNG wire#w1
      I_Contact( #"iSafetyGate Opened Monitor" )
      I_Contact( #ioSafetyGateLock )
      wire#w4
      S_Coil( #"sSafetyGate LockRequest" )
   END_RUNG
   RUNG wire#w4
      R_Coil( #"sSafetyGate UnlockRequest" )
   END_RUNG
   // the same network as SCL:
   #_w1 := #ioHMI_Interface.CMD.RequestPB AND NOT #sP_Trig[1];   // rising edge
   #sP_Trig[1] := #ioHMI_Interface.CMD.RequestPB;
   #_w2 := #_w1 AND #iSysInface.ManualMode;
   IF #_w2 AND (NOT #"iSafetyGate Opened Monitor" OR #"iSafetyGate Opened Monitor") AND #ioSafetyGateLock THEN
       #"sSafetyGate UnlockRequest" := TRUE;
       #"sSafetyGate LockRequest" := FALSE;
   END_IF;
   IF #_w2 AND NOT #"iSafetyGate Opened Monitor" AND NOT #ioSafetyGateLock THEN
       #"sSafetyGate LockRequest" := TRUE;
       #"sSafetyGate UnlockRequest" := FALSE;
   END_IF;
END_REGION

REGION Network 4: 安全门开门请求标志位 / Safety door opening request flag bit
   RUNG wire#powerrail
      Contact( #tAlyways_On )
      wire#w1
      I_Contact( #iSysInface.ManualMode )
      { S7_Templates := "SrcType := Int" } NE_Contact(in1 := #iMode, in2 := 2)
      R_Coil( #"sSafetyGate UnlockRequest" )
   END_RUNG
   RUNG wire#w1
      Contact( #iSysInface.ManualMode )
      P_Trig( #sP_Trig[2] )
      wire#w2
      R_Coil( #"sSafetyGate UnlockRequest" )
   END_RUNG
   RUNG wire#w2
      R_Coil( #"sSafetyGate LockRequest" )
   END_RUNG
   RUNG wire#w1
      Contact( #ioSafetyGateLock )
      wire#w3
      N_Trig( #sN_Trig[1] )
      R_Coil( #"sSafetyGate UnlockRequest" )
   END_RUNG
   RUNG wire#w3
      P_Trig( #sP_Trig[3] )
      R_Coil( #"sSafetyGate LockRequest" )
   END_RUNG
   // the same network as SCL:
   IF #tAlyways_On AND NOT #iSysInface.ManualMode AND (#iMode <> 2) THEN
       #"sSafetyGate UnlockRequest" := FALSE;
   END_IF;
   #_w1 := #tAlyways_On AND #iSysInface.ManualMode;
   #_w2 := #_w1 AND NOT #sP_Trig[2];   // rising edge
   #sP_Trig[2] := #_w1;
   IF #_w2 THEN
       #"sSafetyGate UnlockRequest" := FALSE;
       #"sSafetyGate LockRequest" := FALSE;
   END_IF;
   #_w3 := #tAlyways_On AND #ioSafetyGateLock;
   #_w4 := NOT #_w3 AND #sN_Trig[1];   // falling edge
   #sN_Trig[1] := #_w3;
   IF #_w4 THEN #"sSafetyGate UnlockRequest" := FALSE; END_IF;
   #_w5 := #_w3 AND NOT #sP_Trig[3];   // rising edge
   #sP_Trig[3] := #_w3;
   IF #_w5 THEN #"sSafetyGate LockRequest" := FALSE; END_IF;
END_REGION

REGION Network 5: Reset SafetyGateLock
   // 安全门解锁
   RUNG wire#powerrail
      Contact( #iSysInface.ManualMode )
      Contact( #"sSafetyGate UnlockRequest" )
      wire#w1
      I_Contact( #"iSafetyGate Opened Monitor" )
      wire#w2
      R_Coil( #ioSafetyGateLock )
   END_RUNG
   RUNG wire#w1
      Contact( #"iSafetyGate Opened Monitor" )
   END_RUNG wire#w2
   RUNG wire#powerrail
      Contact( #iSysInface.Auto.Mode )
      { S7_Templates := "SrcType := Int" } EQ_Contact(in1 := #iMode, in2 := 2)
      Contact( #"sSafetyGate UnlockRequest" )
   END_RUNG wire#w2
   // the same network as SCL:
   IF (#iSysInface.ManualMode AND #"sSafetyGate UnlockRequest" AND (NOT #"iSafetyGate Opened Monitor" OR #"iSafetyGate Opened Monitor")) OR (#iSysInface.Auto.Mode AND (#iMode = 2) AND #"sSafetyGate UnlockRequest") THEN
       #ioSafetyGateLock := FALSE;
   END_IF;
END_REGION

REGION Network 6: Set SafetyGate Lock
   // 安全门锁定
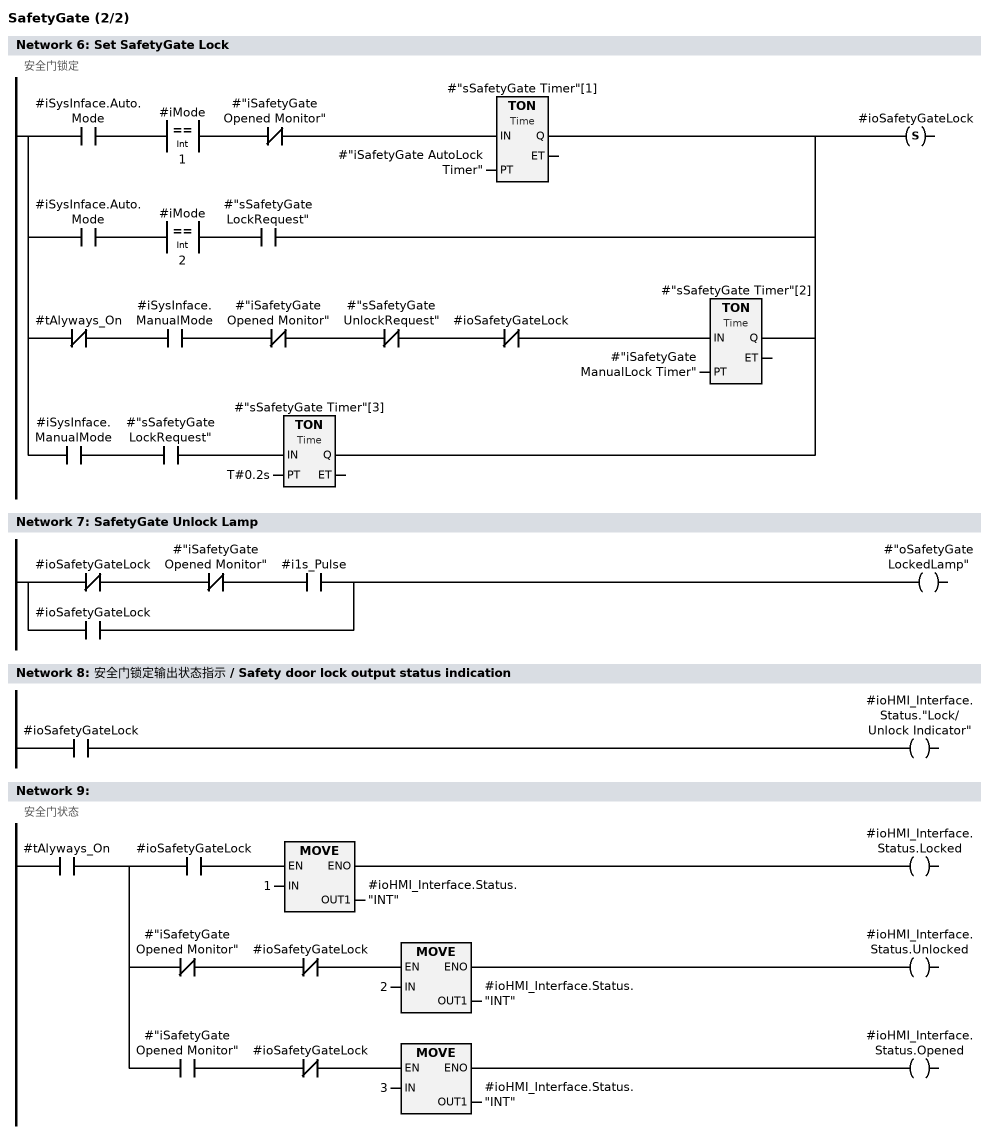
   RUNG wire#powerrail
      Contact( #iSysInface.Auto.Mode )
      { S7_Templates := "SrcType := Int" } EQ_Contact(in1 := #iMode, in2 := 1)
      I_Contact( #"iSafetyGate Opened Monitor" )
      { S7_Templates := "time_type := Time" } #"sSafetyGate Timer"[1].TON(pt := #"iSafetyGate AutoLock Timer", et =>)
      wire#w1
      S_Coil( #ioSafetyGateLock )
   END_RUNG
   RUNG wire#powerrail
      Contact( #iSysInface.Auto.Mode )
      { S7_Templates := "SrcType := Int" } EQ_Contact(in1 := #iMode, in2 := 2)
      Contact( #"sSafetyGate LockRequest" )
   END_RUNG wire#w1
   RUNG wire#powerrail
      I_Contact( #tAlyways_On )
      Contact( #iSysInface.ManualMode )
      I_Contact( #"iSafetyGate Opened Monitor" )
      I_Contact( #"sSafetyGate UnlockRequest" )
      I_Contact( #ioSafetyGateLock )
      { S7_Templates := "time_type := Time" } #"sSafetyGate Timer"[2].TON(pt := #"iSafetyGate ManualLock Timer", et =>)
   END_RUNG wire#w1
   RUNG wire#powerrail
      Contact( #iSysInface.ManualMode )
      Contact( #"sSafetyGate LockRequest" )
      { S7_Templates := "time_type := Time" } #"sSafetyGate Timer"[3].TON(pt := T#0.2s, et =>)
   END_RUNG wire#w1
   // the same network as SCL:
   #"sSafetyGate Timer"[1].TON(IN := #iSysInface.Auto.Mode AND (#iMode = 1) AND NOT #"iSafetyGate Opened Monitor",
                           PT := #"iSafetyGate AutoLock Timer");
   #_w1 := #"sSafetyGate Timer"[1].Q;
   #"sSafetyGate Timer"[2].TON(IN := NOT #tAlyways_On AND #iSysInface.ManualMode AND NOT #"iSafetyGate Opened Monitor" AND NOT #"sSafetyGate UnlockRequest" AND NOT #ioSafetyGateLock,
                           PT := #"iSafetyGate ManualLock Timer");
   #_w2 := #"sSafetyGate Timer"[2].Q;
   #"sSafetyGate Timer"[3].TON(IN := #iSysInface.ManualMode AND #"sSafetyGate LockRequest", PT := T#0.2s);
   IF #_w1 OR (#iSysInface.Auto.Mode AND (#iMode = 2) AND #"sSafetyGate LockRequest") OR #_w2 OR #"sSafetyGate Timer"[3].Q THEN
       #ioSafetyGateLock := TRUE;
   END_IF;
END_REGION

REGION Network 7: SafetyGate Unlock Lamp
   RUNG wire#powerrail
      I_Contact( #ioSafetyGateLock )
      I_Contact( #"iSafetyGate Opened Monitor" )
      Contact( #i1s_Pulse )
      wire#w1
      Coil( #"oSafetyGate LockedLamp" )
   END_RUNG
   RUNG wire#powerrail
      Contact( #ioSafetyGateLock )
   END_RUNG wire#w1
   // the same network as SCL:
   #"oSafetyGate LockedLamp" := (NOT #ioSafetyGateLock AND NOT #"iSafetyGate Opened Monitor" AND #i1s_Pulse) OR #ioSafetyGateLock;
END_REGION

REGION Network 8: 安全门锁定输出状态指示 / Safety door lock output status indication
   RUNG wire#powerrail
      Contact( #ioSafetyGateLock )
      Coil( #ioHMI_Interface.Status."Lock/Unlock Indicator" )
   END_RUNG
   // the same network as SCL:
   #ioHMI_Interface.Status."Lock/Unlock Indicator" := #ioSafetyGateLock;
END_REGION

REGION Network 9
   // 安全门状态
   RUNG wire#powerrail
      Contact( #tAlyways_On )
      wire#w1
      Contact( #ioSafetyGateLock )
      Move(in := 1, out1 => #ioHMI_Interface.Status."INT")
      Coil( #ioHMI_Interface.Status.Locked )
   END_RUNG
   RUNG wire#w1
      I_Contact( #"iSafetyGate Opened Monitor" )
      I_Contact( #ioSafetyGateLock )
      Move(in := 2, out1 => #ioHMI_Interface.Status."INT")
      Coil( #ioHMI_Interface.Status.Unlocked )
   END_RUNG
   RUNG wire#w1
      Contact( #"iSafetyGate Opened Monitor" )
      I_Contact( #ioSafetyGateLock )
      Move(in := 3, out1 => #ioHMI_Interface.Status."INT")
      Coil( #ioHMI_Interface.Status.Opened )
   END_RUNG
   // the same network as SCL:
   #_w1 := #tAlyways_On AND #ioSafetyGateLock;
   IF #_w1 THEN #ioHMI_Interface.Status."INT" := 1; END_IF;
   #ioHMI_Interface.Status.Locked := #_w1;
   #_w2 := #tAlyways_On AND NOT #"iSafetyGate Opened Monitor" AND NOT #ioSafetyGateLock;
   IF #_w2 THEN #ioHMI_Interface.Status."INT" := 2; END_IF;
   #ioHMI_Interface.Status.Unlocked := #_w2;
   #_w3 := #tAlyways_On AND #"iSafetyGate Opened Monitor" AND NOT #ioSafetyGateLock;
   IF #_w3 THEN #ioHMI_Interface.Status."INT" := 3; END_IF;
   #ioHMI_Interface.Status.Opened := #_w3;
END_REGION
END_FUNCTION_BLOCK

FUNCTION "ST10_PartData" : Void   // FC1500, SCL
{ S7_Optimized_Access := 'TRUE' }
// stored: SetENOAutomatically false
   VAR_INPUT
      iSysMode : "RCS_SysComInterface_V1";
   END_VAR
   VAR_TEMP
      idex : Int;
   END_VAR
BEGIN
END_FUNCTION

FUNCTION "ST10_Analog" : Void   // FC1080, SCL
{ S7_Optimized_Access := 'TRUE' }
// stored: AutoNumber false, SetENOAutomatically false
   VAR_INPUT
      iSysMode : "RCS_SysComInterface_V1";
   END_VAR
   VAR_TEMP
      idex : Int;
   END_VAR
BEGIN


   REGION 氮气压模拟量
       //定义编号
       #idex := 1;
       //功能块调用

    END_REGION
END_FUNCTION

FUNCTION "CuringOven" : Void   // FC900, LAD
{ S7_Optimized_Access := 'TRUE' }
// stored: AutoNumber false, SetENOAutomatically false
BEGIN

REGION Network 1
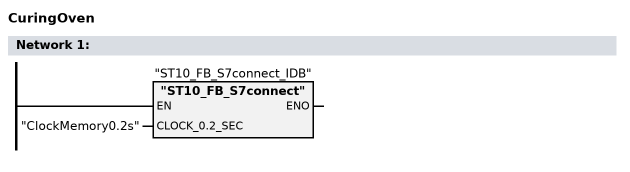
   RUNG wire#powerrail
      "ST10_FB_S7connect_IDB"("CLOCK_0.2_SEC" := "ClockMemory0.2s")
   END_RUNG
   // the same network as SCL:
   "ST10_FB_S7connect_IDB"("CLOCK_0.2_SEC" := "ClockMemory0.2s");   // "ST10_FB_S7connect"
END_REGION
END_FUNCTION

FUNCTION_BLOCK "ST10_FB_S7connect"   // FB900, LAD
{ S7_Optimized_Access := 'TRUE' }
// stored: AutoNumber false, MemoryReserve 100, SetENOAutomatically false
   VAR_INPUT
      "CLOCK_0.2_SEC" : Bool;
   END_VAR
   VAR
      Always_On : Bool;
      Status_Get : Array[1..6] of Struct
         NDR : Bool;
         Error : Bool;
         Status : Int;
      END_STRUCT;
      Status_Put : Array[1..6] of Struct
         Done : Bool;
         Error : Bool;
         Status : Int;
      END_STRUCT;
      GET_Instance1 { S7_SetPoint := 'True'} : GET;
      GET_Instance2 { S7_SetPoint := 'True'} : GET;
      PUT_Instance1 { S7_SetPoint := 'True'} : PUT;
      PUT_Instance2 { S7_SetPoint := 'True'} : PUT;
      PLs { S7_SetPoint := 'True'} : Array[1..6] of Bool;
   END_VAR
   VAR DB_SPECIFIC
      TON : Array[1..5] of TON_TIME;
   END_VAR
   VAR
      NextStation_OffLine : Bool;   // S7心跳超时
   END_VAR
BEGIN

REGION Network 1: **************** 和40交互 **************** / **************** ****************
END_REGION

REGION Network 2: PUT
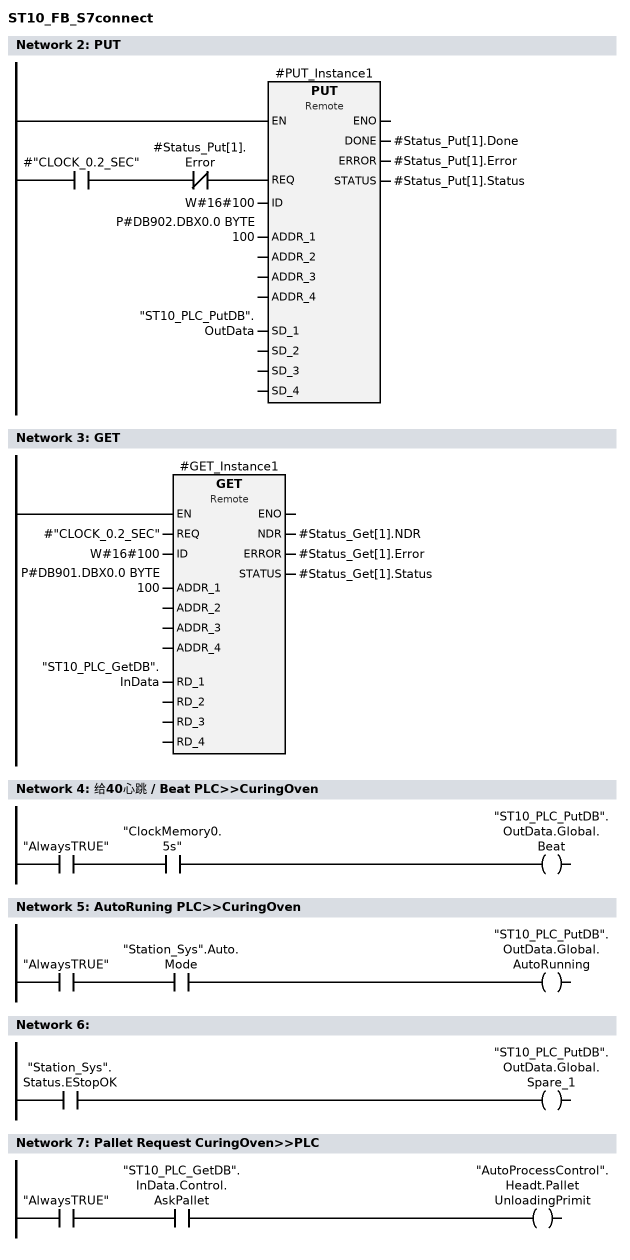
   RUNG wire#powerrail
      { S7_Templates := "[remote_type := Remote, local_type := Variant]" } #PUT_Instance1.PUT(REQ := wire#w1, ID := W#16#100, ADDR_1 := P#DB902.DBX0.0 BYTE 100, ADDR_2 :=, ADDR_3 :=, ADDR_4 :=, SD_1 := "ST10_PLC_PutDB".OutData, SD_2 :=, SD_3 :=, SD_4 :=, DONE => #Status_Put[1].Done, ERROR => #Status_Put[1].Error, STATUS => #Status_Put[1].Status)
   END_RUNG
   RUNG wire#powerrail
      Contact( #"CLOCK_0.2_SEC" )
      I_Contact( #Status_Put[1].Error )
   END_RUNG wire#w1
   // the same network as SCL:
   #PUT_Instance1(REQ := #"CLOCK_0.2_SEC" AND NOT #Status_Put[1].Error,   // PUT
                  ID := W#16#100,
                  ADDR_1 := P#DB902.DBX0.0 BYTE 100,
                  SD_1 := "ST10_PLC_PutDB".OutData,
                  DONE => #Status_Put[1].Done,
                  ERROR => #Status_Put[1].Error,
                  STATUS => #Status_Put[1].Status);
END_REGION

REGION Network 3: GET
   RUNG wire#powerrail
      { S7_Templates := "[remote_type := Remote, local_type := Variant]" } #GET_Instance1.GET(REQ := #"CLOCK_0.2_SEC", ID := W#16#100, ADDR_1 := P#DB901.DBX0.0 BYTE 100, ADDR_2 :=, ADDR_3 :=, ADDR_4 :=, RD_1 := "ST10_PLC_GetDB".InData, RD_2 :=, RD_3 :=, RD_4 :=, NDR => #Status_Get[1].NDR, ERROR => #Status_Get[1].Error, STATUS => #Status_Get[1].Status)
   END_RUNG
   // the same network as SCL:
   #GET_Instance1(REQ := #"CLOCK_0.2_SEC",   // GET
                  ID := W#16#100,
                  ADDR_1 := P#DB901.DBX0.0 BYTE 100,
                  RD_1 := "ST10_PLC_GetDB".InData,
                  NDR => #Status_Get[1].NDR,
                  ERROR => #Status_Get[1].Error,
                  STATUS => #Status_Get[1].Status);
END_REGION

REGION Network 4: 给40心跳 / Beat PLC>>CuringOven
   RUNG wire#powerrail
      Contact( "AlwaysTRUE" )
      Contact( "ClockMemory0.5s" )
      Coil( "ST10_PLC_PutDB".OutData.Global.Beat )
   END_RUNG
   // the same network as SCL:
   "ST10_PLC_PutDB".OutData.Global.Beat := "AlwaysTRUE" AND "ClockMemory0.5s";
END_REGION

REGION Network 5: AutoRuning PLC>>CuringOven
   RUNG wire#powerrail
      Contact( "AlwaysTRUE" )
      Contact( "Station_Sys".Auto.Mode )
      Coil( "ST10_PLC_PutDB".OutData.Global.AutoRunning )
   END_RUNG
   // the same network as SCL:
   "ST10_PLC_PutDB".OutData.Global.AutoRunning := "AlwaysTRUE" AND "Station_Sys".Auto.Mode;
END_REGION

REGION Network 6
   RUNG wire#powerrail
      Contact( "Station_Sys".Status.EStopOK )
      Coil( "ST10_PLC_PutDB".OutData.Global.Spare_1 )
   END_RUNG
   // the same network as SCL:
   "ST10_PLC_PutDB".OutData.Global.Spare_1 := "Station_Sys".Status.EStopOK;
END_REGION

REGION Network 7: Pallet Request CuringOven>>PLC
   RUNG wire#powerrail
      Contact( "AlwaysTRUE" )
      Contact( "ST10_PLC_GetDB".InData.Control.AskPallet )
      Coil( "AutoProcessControl".Headt.PalletUnloadingPrimit )
   END_RUNG
   // the same network as SCL:
   "AutoProcessControl".Headt.PalletUnloadingPrimit := "AlwaysTRUE" AND "ST10_PLC_GetDB".InData.Control.AskPallet;
END_REGION
END_FUNCTION_BLOCK

FUNCTION "IV3" : Void   // FC2100, LAD
{ S7_Optimized_Access := 'TRUE' }
// stored: AutoNumber false, SetENOAutomatically false
BEGIN

REGION Network 1: IV3
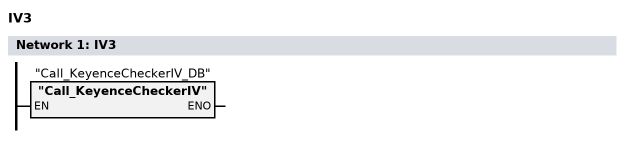
   RUNG wire#powerrail
      "Call_KeyenceCheckerIV_DB"()
   END_RUNG
   // the same network as SCL:
   "Call_KeyenceCheckerIV_DB"();   // "Call_KeyenceCheckerIV"
END_REGION
END_FUNCTION

FUNCTION_BLOCK "Call_KeyenceCheckerIV"   // FB2100, SCL
{ S7_Optimized_Access := 'TRUE' }
// stored: AutoNumber false, MemoryReserve 100, SetENOAutomatically false
   VAR
      InsKeyenceCheckerIV3810A1 : "FB_KeyenceCheckerIV3";   // 声明相机功能块的实例
      InsKeyenceCheckerIV3811A1 : "FB_KeyenceCheckerIV3";   // 声明相机功能块的实例
      nIndex { S7_SetPoint := 'True'} : Int;
   END_VAR
BEGIN

   //810A1
   REGION KeyenceCheckerIV3() 

       REGION HardwareConfigGuidance()
           // 组态说明/Hardware config Guidance
           // 输入/Input
           // Command Status Bits_1
           // Device Result Bits_1
           // Device Status Words_1
           // Device Statistics_1
           // Position Adjust Result_1
           // Tool Result_1
           // Tool Result_2
           // 输出/Output
           // Command Control_1
       END_REGION

       REGION DeviceControl()
           //************************************************************************************************ 
           //设备控制/Device control 
           //************************************************************************************************ 
           //Set device number
           #nIndex := 1;//(For example Constant:ST01_CHECKER_FUNCTION)

           REGION WorkflowControl()
               //************************************************************************************************ 
               //流程控制/Workflow control
               //************************************************************************************************ 
               //---set program number
               //   "DB_KeyenceCheckerIV2".aDev[#nIndex].Out.CommandControl.nProgramNo
               //---set command mode and wait for mode to "MODE_CHECKER_IDLE"
               //   "DB_KeyenceCheckerIV2".aDev[#nIndex].Common.nMode
           END_REGION

           REGION GeneralControl()
               //************************************************************************************************ 
               //常规控制/General control 
               //************************************************************************************************ 
               //Set common parameter
               "DB_KeyenceCheckerIV3".aDev[#nIndex].Common.bScreenActive := "Station_Sys".Manual.Mode;
               "DB_KeyenceCheckerIV3".aDev[#nIndex].Common.bReset := "Station_Sys".Cmd.Reset;
               "DB_KeyenceCheckerIV3".aDev[#nIndex].Common.tMaxProcessTime := t#30s;
           END_REGION

           REGION ParameterConfig()
               //************************************************************************************************ 
               //参数配置/Parameter config 
               //************************************************************************************************ 
           END_REGION

           REGION ModeControl()
               //************************************************************************************************ 
               //设备启动停止/Device mode control
               //************************************************************************************************ 
               // IF NOT "Station_Sys".Status.Run THEN
               //     "DB_KeyenceCheckerIV3".aDev[#nIndex].Common.nMode := 0;
               // END_IF;

               IF "Station_Sys".Manual.Mode THEN
                   "DB_KeyenceCheckerIV3".aDev[#nIndex].Common.nModeSwitch := "MS_MANUAL";
               ELSIF "Station_Sys".Auto.Mode THEN
                   "DB_KeyenceCheckerIV3".aDev[#nIndex].Common.nModeSwitch:=  "MS_Auto";
               ELSE
                   "DB_KeyenceCheckerIV3".aDev[#nIndex].Common.nModeSwitch := "MS_EMPTY";
               END_IF;
               END_REGION

           REGION ConditionControl()
               //************************************************************************************************ 
               //使能控制/Condition control
               //************************************************************************************************ 
               //according to detail information in different use to fill in start condition
               "DB_KeyenceCheckerIV3".aDev[#nIndex].Common.bEnable := "Station_Sys".Status.Run;
           END_REGION

       END_REGION

       REGION HardwareInput()
           //************************************************************************************************ 
           //硬件输入/Hardware input 
           //************************************************************************************************ 
       END_REGION

       REGION CallFunctionBlock()
           //************************************************************************************************
           //功能块调用/Call function block
           //************************************************************************************************
           //according to hardware configuration to type in hardware address

           #InsKeyenceCheckerIV3810A1(#nIndex);


       END_REGION

       REGION HardwareOutput()
           //************************************************************************************************ 
           //硬件输出/Hardware output 
           //************************************************************************************************ 
       END_REGION

   END_REGION


   //811A1
   REGION KeyenceCheckerIV3() 

       REGION HardwareConfigGuidance()
           // 组态说明/Hardware config Guidance
           // 输入/Input
           // Command Status Bits_1
           // Device Result Bits_1
           // Device Status Words_1
           // Device Statistics_1
           // Position Adjust Result_1
           // Tool Result_1
           // Tool Result_2
           // 输出/Output
           // Command Control_1
       END_REGION

       REGION DeviceControl()
           //************************************************************************************************ 
           //设备控制/Device control 
           //************************************************************************************************ 
           //Set device number
           #nIndex := 2;//(For example Constant:ST01_CHECKER_FUNCTION)

           REGION WorkflowControl()
               //************************************************************************************************ 
               //流程控制/Workflow control
               //************************************************************************************************ 
               //---set program number
               //   "DB_KeyenceCheckerIV2".aDev[#nIndex].Out.CommandControl.nProgramNo
               //---set command mode and wait for mode to "MODE_CHECKER_IDLE"
               //   "DB_KeyenceCheckerIV2".aDev[#nIndex].Common.nMode
           END_REGION

           REGION GeneralControl()
               //************************************************************************************************ 
               //常规控制/General control 
               //************************************************************************************************ 
               //Set common parameter
               "DB_KeyenceCheckerIV3".aDev[#nIndex].Common.bScreenActive := "Station_Sys".Manual.Mode;
               "DB_KeyenceCheckerIV3".aDev[#nIndex].Common.bReset := "Station_Sys".Cmd.Reset;
               "DB_KeyenceCheckerIV3".aDev[#nIndex].Common.tMaxProcessTime := t#30s;
           END_REGION

           REGION ParameterConfig()
               //************************************************************************************************ 
               //参数配置/Parameter config 
               //************************************************************************************************ 
           END_REGION

           REGION ModeControl()
               //************************************************************************************************ 
               //设备启动停止/Device mode control
               //************************************************************************************************ 
               // IF NOT "Station_Sys".Status.Run THEN
               //     "DB_KeyenceCheckerIV3".aDev[#nIndex].Common.nMode := 0;
               // END_IF;

               IF "Station_Sys".Manual.Mode THEN
                   "DB_KeyenceCheckerIV3".aDev[#nIndex].Common.nModeSwitch := "MS_MANUAL";
               ELSIF "Station_Sys".Auto.Mode THEN
                   "DB_KeyenceCheckerIV3".aDev[#nIndex].Common.nModeSwitch := "MS_Auto";
               ELSE
                   "DB_KeyenceCheckerIV3".aDev[#nIndex].Common.nModeSwitch := "MS_EMPTY";
               END_IF;
           END_REGION

           REGION ConditionControl()
               //************************************************************************************************ 
               //使能控制/Condition control
               //************************************************************************************************ 
               //according to detail information in different use to fill in start condition
               "DB_KeyenceCheckerIV3".aDev[#nIndex].Common.bEnable := "Station_Sys".Status.Run;
           END_REGION

       END_REGION

       REGION HardwareInput()
           //************************************************************************************************ 
           //硬件输入/Hardware input 
           //************************************************************************************************ 
       END_REGION

       REGION CallFunctionBlock()
           //************************************************************************************************
           //功能块调用/Call function block
           //************************************************************************************************
           //according to hardware configuration to type in hardware address

           #InsKeyenceCheckerIV3811A1(#nIndex);


       END_REGION

       REGION HardwareOutput()
           //************************************************************************************************ 
           //硬件输出/Hardware output 
           //************************************************************************************************ 
       END_REGION

   END_REGION
END_FUNCTION_BLOCK

FUNCTION_BLOCK "FB_KeyenceCheckerIV3"
{ S7_Optimized_Access := 'TRUE' }
VERSION : 0.1
// ATTRIBUTES
// AUTO_NUMBER = False
// BLOCK_NUMBER = 2101
// END_ATTRIBUTES
   VAR_INPUT 
      I_nID : Int;
   END_VAR

   VAR 
      rtrigManualMode {InstructionName := 'R_TRIG'; LibVersion := '1.0'} : R_TRIG;
      ftrigManualMode {InstructionName := 'F_TRIG'; LibVersion := '1.0'} : F_TRIG;
      "****Common*******" : Bool;
      nStep : Int;
      nNextStep : Int;
      nLastStep : Int;
      bCondition : Bool;
      fbNextstep { S7_SetPoint := 'False'} : "FB_Next";
      tonProcessOvertime {InstructionName := 'TON_TIME'; LibVersion := '1.0'; S7_SetPoint := 'False'} : TON_TIME;
      "****Local******" : Bool;
      aToolResultReset : Array[1..64] of Bool;
      ToolResultResult : Array[1..64] of Struct
         nToolMatchingRate : Word;
         nToolMatchingRateMAX : Word;
         nToolMatchingRateMIN : Word;
         nToolLowerLimitValue : Word;
         nToolUpperLimitValue : Word;
         nDecimalPosition : Word;
         "nPitchPresentValueMAX/ColorAverageH (hue)" : Word;
         "nPitchPresentValueMIN/ColorAverageS(saturation)" : Word;
         "nNumberOfPitches/ColorAverageV(brightness)/BrightnessAverage" : Word;
         nReserved1 : Word;
      END_STRUCT;
      bCompleteToggleSign : Bool;
      rtrigCompleteToggle {InstructionName := 'R_TRIG'; LibVersion := '1.0'; S7_SetPoint := 'False'} : R_TRIG;
      ftrigCompleteToggle {InstructionName := 'F_TRIG'; LibVersion := '1.0'; S7_SetPoint := 'False'} : F_TRIG;
      nIdx : Int;
      nTriggerFailCount : Byte;
      "****Instruction******" : Bool;
   END_VAR
   VAR DB_SPECIFIC
      nWord : Word;
      aWord { ExternalAccessible := 'False'; ExternalVisible := 'False'; ExternalWritable := 'False'} AT nWord : Array[0..1] of Byte;
      nDWord : DWord;
      aDWord { ExternalAccessible := 'False'; ExternalVisible := 'False'; ExternalWritable := 'False'} AT nDWord : Array[0..3] of Byte;
   END_VAR
   VAR 
      nIndex3 : Int;
   END_VAR

   VAR_TEMP 
      nByte : Byte;
      aInput_Byte1 : Array[0..3] of Byte;
      aInput_Byte2 : Array[0..3] of Byte;
      aInput_Byte3 : Array[0..15] of Byte;
      aInput_Byte4 : Array[0..27] of Byte;
      aInput_Byte5 : Array[0..19] of Byte;
      aInput_Byte6 : Array[0..63] of Struct
         bInput_Byte0 : Byte;
         bInput_Byte1 : Byte;
         bInput_Byte2 : Byte;
         bInput_Byte3 : Byte;
         bInput_Byte4 : Byte;
         bInput_Byte5 : Byte;
         bInput_Byte6 : Byte;
         bInput_Byte7 : Byte;
         bInput_Byte8 : Byte;
         bInput_Byte9 : Byte;
         bInput_Byte10 : Byte;
         bInput_Byte11 : Byte;
         bInput_Byte12 : Byte;
         bInput_Byte13 : Byte;
         bInput_Byte14 : Byte;
         bInput_Byte15 : Byte;
         bInput_Byte16 : Byte;
         bInput_Byte17 : Byte;
         bInput_Byte18 : Byte;
         bInput_Byte19 : Byte;
      END_STRUCT;
      aInput_Byte7 : Array[0..7] of Byte;
      aOutput_Byte1 : Array[0..11] of Byte;
      aRetvalRead : Array[1..22] of Int;
      aRetvalWrite : Array[1..1] of Int;
   END_VAR

   VAR CONSTANT 
      MODE_CHECKER_IDLE : Int := 0;
      MODE_CHECKER_START : Int := 1;
      MODE_CHECKER_REGISTER : Int := 4;
      MODE_CHECKER_CLEAR : Int := 5;
      MODE_CHECKER_RESET : Int := 99;
   END_VAR


BEGIN
	(*
	=============================================================================
	BBSS Automation
	(c)Copyright 2022 All Rights Reserved
	-----------------------------------------------------------------------------
	Functionality:
	This function block manager keyence checker iv3 control
	-----------------------------------------------------------------------------
	Change log table:
	Version   Date Y/M/D    Person       Description
	3.0.1     21/09/01      Xiangxiang   Active simulation
	3.0.4     22/01/20      Yuan Li      Handshake disabled
	3.0.5     22/05/13      Xuecao Guo   Update IV2 to IV3
	4.0.0     22/08/18      Huiyun       Separate condition and definition
	=============================================================================
	*)
	
	REGION ReadData()
	    //************************************************************************************************ 
	    //从接口读取数据/Read data from interface
	    //************************************************************************************************ 
	    //命令状态/Command Status bits
	    #aRetvalRead[1] := DPRD_DAT(LADDR := "DB_KeyenceCheckerIV3".aDev[#I_nID].Para.nInAdr1, RECORD => #aInput_Byte1);
	    //设备结果/Device Results bits
	    #aRetvalRead[2] := DPRD_DAT(LADDR := "DB_KeyenceCheckerIV3".aDev[#I_nID].Para.nInAdr2, RECORD => #aInput_Byte2);
	    //设备状态/Device status words
	    #aRetvalRead[3] := DPRD_DAT(LADDR := "DB_KeyenceCheckerIV3".aDev[#I_nID].Para.nInAdr3, RECORD => #aInput_Byte3);
	    //设备统计/Device statistics
	    #aRetvalRead[4] := DPRD_DAT(LADDR := "DB_KeyenceCheckerIV3".aDev[#I_nID].Para.nInAdr4, RECORD => #aInput_Byte4);
	    //位置修正结果/Position adjust result
	    #aRetvalRead[5] := DPRD_DAT(LADDR := "DB_KeyenceCheckerIV3".aDev[#I_nID].Para.nInAdr5, RECORD => #aInput_Byte5);
	    //工具1处理结果/Tool1 result
	    #aRetvalRead[6] := DPRD_DAT(LADDR := "DB_KeyenceCheckerIV3".aDev[#I_nID].Para.nInAdr6, RECORD => #aInput_Byte6[0]);
	    //工具2处理结果/Tool2 result
	    #aRetvalRead[7] := DPRD_DAT(LADDR := "DB_KeyenceCheckerIV3".aDev[#I_nID].Para.nInAdr7, RECORD => #aInput_Byte6[1]);
	    //工具3处理结果/Tool3 result
	    #aRetvalRead[8] := DPRD_DAT(LADDR := "DB_KeyenceCheckerIV3".aDev[#I_nID].Para.nInAdr8, RECORD => #aInput_Byte6[2]);
	    //工具4处理结果/Tool4 result
	    #aRetvalRead[9] := DPRD_DAT(LADDR := "DB_KeyenceCheckerIV3".aDev[#I_nID].Para.nInAdr9, RECORD => #aInput_Byte6[3]);
	    //工具5处理结果/Tool5 result
	    #aRetvalRead[10] := DPRD_DAT(LADDR := "DB_KeyenceCheckerIV3".aDev[#I_nID].Para.nInAdr10, RECORD => #aInput_Byte6[4]);
	    //工具6处理结果/Tool6 result
	    #aRetvalRead[11] := DPRD_DAT(LADDR := "DB_KeyenceCheckerIV3".aDev[#I_nID].Para.nInAdr11, RECORD => #aInput_Byte6[5]);
	    //工具7处理结果/Tool7 result
	    #aRetvalRead[12] := DPRD_DAT(LADDR := "DB_KeyenceCheckerIV3".aDev[#I_nID].Para.nInAdr12, RECORD => #aInput_Byte6[6]);
	    //工具8处理结果/Tool8 result
	    #aRetvalRead[13] := DPRD_DAT(LADDR := "DB_KeyenceCheckerIV3".aDev[#I_nID].Para.nInAdr13, RECORD => #aInput_Byte6[7]);
	    //工具9处理结果/Tool9 result
	    #aRetvalRead[14] := DPRD_DAT(LADDR := "DB_KeyenceCheckerIV3".aDev[#I_nID].Para.nInAdr14, RECORD => #aInput_Byte6[8]);
	    //工具10处理结果/Tool10 result
	    #aRetvalRead[15] := DPRD_DAT(LADDR := "DB_KeyenceCheckerIV3".aDev[#I_nID].Para.nInAdr15, RECORD => #aInput_Byte6[9]);
	    //工具11处理结果/Tool11 result
	    #aRetvalRead[16] := DPRD_DAT(LADDR := "DB_KeyenceCheckerIV3".aDev[#I_nID].Para.nInAdr16, RECORD => #aInput_Byte6[10]);
	    //工具12处理结果/Tool12 result
	    #aRetvalRead[17] := DPRD_DAT(LADDR := "DB_KeyenceCheckerIV3".aDev[#I_nID].Para.nInAdr17, RECORD => #aInput_Byte6[11]);
	    //工具13处理结果/Tool13 result
	    #aRetvalRead[18] := DPRD_DAT(LADDR := "DB_KeyenceCheckerIV3".aDev[#I_nID].Para.nInAdr18, RECORD => #aInput_Byte6[12]);
	    //工具14处理结果/Tool14 result
	    #aRetvalRead[19] := DPRD_DAT(LADDR := "DB_KeyenceCheckerIV3".aDev[#I_nID].Para.nInAdr19, RECORD => #aInput_Byte6[13]);
	    //工具15处理结果/Tool15 result
	    #aRetvalRead[20] := DPRD_DAT(LADDR := "DB_KeyenceCheckerIV3".aDev[#I_nID].Para.nInAdr20, RECORD => #aInput_Byte6[14]);
	    //工具16处理结果/Tool16 result
	    #aRetvalRead[21] := DPRD_DAT(LADDR := "DB_KeyenceCheckerIV3".aDev[#I_nID].Para.nInAdr21, RECORD => #aInput_Byte6[15]);
	    //工具17处理结果/Tool1 result
	    #aRetvalRead[6] := DPRD_DAT(LADDR := "DB_KeyenceCheckerIV3".aDev[#I_nID].Para.nInAdr22, RECORD => #aInput_Byte6[16]);
	    //工具18处理结果/Tool2 result
	    #aRetvalRead[7] := DPRD_DAT(LADDR := "DB_KeyenceCheckerIV3".aDev[#I_nID].Para.nInAdr23, RECORD => #aInput_Byte6[17]);
	    //工具19处理结果/Tool3 result
	    #aRetvalRead[8] := DPRD_DAT(LADDR := "DB_KeyenceCheckerIV3".aDev[#I_nID].Para.nInAdr24, RECORD => #aInput_Byte6[18]);
	    //工具20处理结果/Tool4 result
	    #aRetvalRead[9] := DPRD_DAT(LADDR := "DB_KeyenceCheckerIV3".aDev[#I_nID].Para.nInAdr25, RECORD => #aInput_Byte6[19]);
	    //工具21处理结果/Tool5 result
	    #aRetvalRead[10] := DPRD_DAT(LADDR := "DB_KeyenceCheckerIV3".aDev[#I_nID].Para.nInAdr26, RECORD => #aInput_Byte6[20]);
	    //工具22处理结果/Tool6 result
	    #aRetvalRead[11] := DPRD_DAT(LADDR := "DB_KeyenceCheckerIV3".aDev[#I_nID].Para.nInAdr27, RECORD => #aInput_Byte6[21]);
	    //工具23处理结果/Tool7 result
	    #aRetvalRead[12] := DPRD_DAT(LADDR := "DB_KeyenceCheckerIV3".aDev[#I_nID].Para.nInAdr28, RECORD => #aInput_Byte6[22]);
	    //工具24处理结果/Tool8 result
	    #aRetvalRead[13] := DPRD_DAT(LADDR := "DB_KeyenceCheckerIV3".aDev[#I_nID].Para.nInAdr29, RECORD => #aInput_Byte6[23]);
	    //工具25处理结果/Tool9 result
	    #aRetvalRead[14] := DPRD_DAT(LADDR := "DB_KeyenceCheckerIV3".aDev[#I_nID].Para.nInAdr30, RECORD => #aInput_Byte6[24]);
	    //工具26处理结果/Tool10 result
	    #aRetvalRead[15] := DPRD_DAT(LADDR := "DB_KeyenceCheckerIV3".aDev[#I_nID].Para.nInAdr31, RECORD => #aInput_Byte6[25]);
	    //工具27处理结果/Tool11 result
	    #aRetvalRead[16] := DPRD_DAT(LADDR := "DB_KeyenceCheckerIV3".aDev[#I_nID].Para.nInAdr32, RECORD => #aInput_Byte6[26]);
	    //工具28处理结果/Tool12 result
	    #aRetvalRead[17] := DPRD_DAT(LADDR := "DB_KeyenceCheckerIV3".aDev[#I_nID].Para.nInAdr33, RECORD => #aInput_Byte6[27]);
	    //工具29处理结果/Tool13 result
	    #aRetvalRead[18] := DPRD_DAT(LADDR := "DB_KeyenceCheckerIV3".aDev[#I_nID].Para.nInAdr34, RECORD => #aInput_Byte6[28]);
	    //工具30处理结果/Tool14 result
	    #aRetvalRead[19] := DPRD_DAT(LADDR := "DB_KeyenceCheckerIV3".aDev[#I_nID].Para.nInAdr35, RECORD => #aInput_Byte6[29]);
	    //工具31处理结果/Tool15 result
	    #aRetvalRead[20] := DPRD_DAT(LADDR := "DB_KeyenceCheckerIV3".aDev[#I_nID].Para.nInAdr36, RECORD => #aInput_Byte6[30]);
	    //工具32处理结果/Tool16 result
	    #aRetvalRead[21] := DPRD_DAT(LADDR := "DB_KeyenceCheckerIV3".aDev[#I_nID].Para.nInAdr37, RECORD => #aInput_Byte6[31]);
	    //工具33处理结果/Tool1 result
	    #aRetvalRead[6] := DPRD_DAT(LADDR := "DB_KeyenceCheckerIV3".aDev[#I_nID].Para.nInAdr38, RECORD => #aInput_Byte6[32]);
	    //工具34处理结果/Tool2 result
	    #aRetvalRead[7] := DPRD_DAT(LADDR := "DB_KeyenceCheckerIV3".aDev[#I_nID].Para.nInAdr39, RECORD => #aInput_Byte6[33]);
	    //工具35处理结果/Tool3 result
	    #aRetvalRead[8] := DPRD_DAT(LADDR := "DB_KeyenceCheckerIV3".aDev[#I_nID].Para.nInAdr40, RECORD => #aInput_Byte6[34]);
	    //工具36处理结果/Tool4 result
	    #aRetvalRead[9] := DPRD_DAT(LADDR := "DB_KeyenceCheckerIV3".aDev[#I_nID].Para.nInAdr41, RECORD => #aInput_Byte6[35]);
	    //工具37处理结果/Tool5 result
	    #aRetvalRead[10] := DPRD_DAT(LADDR := "DB_KeyenceCheckerIV3".aDev[#I_nID].Para.nInAdr42, RECORD => #aInput_Byte6[36]);
	    //工具38处理结果/Tool6 result
	    #aRetvalRead[11] := DPRD_DAT(LADDR := "DB_KeyenceCheckerIV3".aDev[#I_nID].Para.nInAdr43, RECORD => #aInput_Byte6[37]);
	    //工具39处理结果/Tool7 result
	    #aRetvalRead[12] := DPRD_DAT(LADDR := "DB_KeyenceCheckerIV3".aDev[#I_nID].Para.nInAdr44, RECORD => #aInput_Byte6[38]);
	    //工具40处理结果/Tool8 result
	    #aRetvalRead[13] := DPRD_DAT(LADDR := "DB_KeyenceCheckerIV3".aDev[#I_nID].Para.nInAdr45, RECORD => #aInput_Byte6[39]);
	    //工具41处理结果/Tool9 result
	    #aRetvalRead[14] := DPRD_DAT(LADDR := "DB_KeyenceCheckerIV3".aDev[#I_nID].Para.nInAdr46, RECORD => #aInput_Byte6[40]);
	    //工具42处理结果/Tool10 result
	    #aRetvalRead[15] := DPRD_DAT(LADDR := "DB_KeyenceCheckerIV3".aDev[#I_nID].Para.nInAdr47, RECORD => #aInput_Byte6[41]);
	    //工具43处理结果/Tool11 result
	    #aRetvalRead[16] := DPRD_DAT(LADDR := "DB_KeyenceCheckerIV3".aDev[#I_nID].Para.nInAdr48, RECORD => #aInput_Byte6[42]);
	    //工具44处理结果/Tool12 result
	    #aRetvalRead[17] := DPRD_DAT(LADDR := "DB_KeyenceCheckerIV3".aDev[#I_nID].Para.nInAdr49, RECORD => #aInput_Byte6[43]);
	    //工具45处理结果/Tool13 result
	    #aRetvalRead[18] := DPRD_DAT(LADDR := "DB_KeyenceCheckerIV3".aDev[#I_nID].Para.nInAdr50, RECORD => #aInput_Byte6[44]);
	    //工具46处理结果/Tool14 result
	    #aRetvalRead[19] := DPRD_DAT(LADDR := "DB_KeyenceCheckerIV3".aDev[#I_nID].Para.nInAdr51, RECORD => #aInput_Byte6[45]);
	    //工具47处理结果/Tool15 result
	    #aRetvalRead[20] := DPRD_DAT(LADDR := "DB_KeyenceCheckerIV3".aDev[#I_nID].Para.nInAdr52, RECORD => #aInput_Byte6[46]);
	    //工具48处理结果/Tool16 result
	    #aRetvalRead[21] := DPRD_DAT(LADDR := "DB_KeyenceCheckerIV3".aDev[#I_nID].Para.nInAdr53, RECORD => #aInput_Byte6[47]);
	    //工具49处理结果/Tool1 result
	    #aRetvalRead[6] := DPRD_DAT(LADDR := "DB_KeyenceCheckerIV3".aDev[#I_nID].Para.nInAdr54, RECORD => #aInput_Byte6[48]);
	    //工具50处理结果/Tool2 result
	    #aRetvalRead[7] := DPRD_DAT(LADDR := "DB_KeyenceCheckerIV3".aDev[#I_nID].Para.nInAdr55, RECORD => #aInput_Byte6[49]);
	    //工具51处理结果/Tool3 result
	    #aRetvalRead[8] := DPRD_DAT(LADDR := "DB_KeyenceCheckerIV3".aDev[#I_nID].Para.nInAdr56, RECORD => #aInput_Byte6[50]);
	    //工具52处理结果/Tool4 result
	    #aRetvalRead[9] := DPRD_DAT(LADDR := "DB_KeyenceCheckerIV3".aDev[#I_nID].Para.nInAdr57, RECORD => #aInput_Byte6[51]);
	    //工具53处理结果/Tool5 result
	    #aRetvalRead[10] := DPRD_DAT(LADDR := "DB_KeyenceCheckerIV3".aDev[#I_nID].Para.nInAdr58, RECORD => #aInput_Byte6[52]);
	    //工具54处理结果/Tool6 result
	    #aRetvalRead[11] := DPRD_DAT(LADDR := "DB_KeyenceCheckerIV3".aDev[#I_nID].Para.nInAdr59, RECORD => #aInput_Byte6[53]);
	    //工具55处理结果/Tool7 result
	    #aRetvalRead[12] := DPRD_DAT(LADDR := "DB_KeyenceCheckerIV3".aDev[#I_nID].Para.nInAdr60, RECORD => #aInput_Byte6[54]);
	    //工具56处理结果/Tool8 result
	    #aRetvalRead[13] := DPRD_DAT(LADDR := "DB_KeyenceCheckerIV3".aDev[#I_nID].Para.nInAdr61, RECORD => #aInput_Byte6[55]);
	    //工具57处理结果/Tool9 result
	    #aRetvalRead[14] := DPRD_DAT(LADDR := "DB_KeyenceCheckerIV3".aDev[#I_nID].Para.nInAdr62, RECORD => #aInput_Byte6[56]);
	    //工具58处理结果/Tool10 result
	    #aRetvalRead[15] := DPRD_DAT(LADDR := "DB_KeyenceCheckerIV3".aDev[#I_nID].Para.nInAdr63, RECORD => #aInput_Byte6[57]);
	    //工具59处理结果/Tool11 result
	    #aRetvalRead[16] := DPRD_DAT(LADDR := "DB_KeyenceCheckerIV3".aDev[#I_nID].Para.nInAdr64, RECORD => #aInput_Byte6[58]);
	    //工具60处理结果/Tool12 result
	    #aRetvalRead[17] := DPRD_DAT(LADDR := "DB_KeyenceCheckerIV3".aDev[#I_nID].Para.nInAdr65, RECORD => #aInput_Byte6[59]);
	    //工具61处理结果/Tool13 result
	    #aRetvalRead[18] := DPRD_DAT(LADDR := "DB_KeyenceCheckerIV3".aDev[#I_nID].Para.nInAdr66, RECORD => #aInput_Byte6[60]);
	    //工具62处理结果/Tool14 result
	    #aRetvalRead[19] := DPRD_DAT(LADDR := "DB_KeyenceCheckerIV3".aDev[#I_nID].Para.nInAdr67, RECORD => #aInput_Byte6[61]);
	    //工具63处理结果/Tool15 result
	    #aRetvalRead[20] := DPRD_DAT(LADDR := "DB_KeyenceCheckerIV3".aDev[#I_nID].Para.nInAdr68, RECORD => #aInput_Byte6[62]);
	    //工具64处理结果/Tool16 result
	    #aRetvalRead[21] := DPRD_DAT(LADDR := "DB_KeyenceCheckerIV3".aDev[#I_nID].Para.nInAdr69, RECORD => #aInput_Byte6[63]);
	    //设备结果/Device Results bits
	    #aRetvalRead[22] := DPRD_DAT(LADDR := "DB_KeyenceCheckerIV3".aDev[#I_nID].Para.nInAdr70, RECORD => #aInput_Byte7);
	    "DB_KeyenceCheckerIV3".aDev[#I_nID].Common.nID := #I_nID;
	END_REGION
	
	REGION CopyReadData()
	    ///************************************************************************************************
	    //分配输入数据/Asignment of the intput data (Statusword)
	    //************************************************************************************************
	    //命令状态/Command status bits
	    //Address 0
	    #nByte := #aInput_Byte1[0];
	    "DB_KeyenceCheckerIV3".aDev[#I_nID].In.CommandStatus.bTriggerResponse := #nByte.%X0;
	    "DB_KeyenceCheckerIV3".aDev[#I_nID].In.CommandStatus.bMasterImageRegistration := #nByte.%X1;
	    "DB_KeyenceCheckerIV3".aDev[#I_nID].In.CommandStatus.bProgramSwitchingResponse := #nByte.%X2;
	    "DB_KeyenceCheckerIV3".aDev[#I_nID].In.CommandStatus.bWarningClearResponse := #nByte.%X3;
	    "DB_KeyenceCheckerIV3".aDev[#I_nID].In.CommandStatus.bStatisticsResetResponse := #nByte.%X4;
	    "DB_KeyenceCheckerIV3".aDev[#I_nID].In.CommandStatus.bBufferClearResponse := #nByte.%X5;
	    "DB_KeyenceCheckerIV3".aDev[#I_nID].In.CommandStatus.bSDCardStopSaveResponse := #nByte.%X6;
	    "DB_KeyenceCheckerIV3".aDev[#I_nID].In.CommandStatus.bChangeParameterResponse := #nByte.%X7;
	    //Address 1
	    #nByte := #aInput_Byte1[1];
	    "DB_KeyenceCheckerIV3".aDev[#I_nID].In.CommandStatus.bTriggerFailed := #nByte.%X0;
	    "DB_KeyenceCheckerIV3".aDev[#I_nID].In.CommandStatus.bMasterImageRegistrationFailed := #nByte.%X1;
	    "DB_KeyenceCheckerIV3".aDev[#I_nID].In.CommandStatus.bProgramSwitchingFailed := #nByte.%X2;
	    "DB_KeyenceCheckerIV3".aDev[#I_nID].In.CommandStatus.bReserved1 := #nByte.%X3;
	    "DB_KeyenceCheckerIV3".aDev[#I_nID].In.CommandStatus.bReserved2 := #nByte.%X4;
	    "DB_KeyenceCheckerIV3".aDev[#I_nID].In.CommandStatus.bReserved3 := #nByte.%X5;
	    "DB_KeyenceCheckerIV3".aDev[#I_nID].In.CommandStatus.bSDCardStopSaveFailed := #nByte.%X6;
	    "DB_KeyenceCheckerIV3".aDev[#I_nID].In.CommandStatus.bChangeParameterFailed := #nByte.%X7;
	    //Address 2 
	    #nByte := #aInput_Byte1[2];
	    "DB_KeyenceCheckerIV3".aDev[#I_nID].In.CommandStatus.bResultAvailable := #nByte.%X0;
	    "DB_KeyenceCheckerIV3".aDev[#I_nID].In.CommandStatus.bResultUpdateComplete := #nByte.%X1;
	    "DB_KeyenceCheckerIV3".aDev[#I_nID].In.CommandStatus.bBusy := #nByte.%X2;
	    "DB_KeyenceCheckerIV3".aDev[#I_nID].In.CommandStatus.bImaging := #nByte.%X3;
	    "DB_KeyenceCheckerIV3".aDev[#I_nID].In.CommandStatus.bRun := #nByte.%X4;
	    "DB_KeyenceCheckerIV3".aDev[#I_nID].In.CommandStatus.bReady := #nByte.%X5;
	    "DB_KeyenceCheckerIV3".aDev[#I_nID].In.CommandStatus.bReserved4 := #nByte.%X6;
	    "DB_KeyenceCheckerIV3".aDev[#I_nID].In.CommandStatus.bSDCardStatus := #nByte.%X7;
	    //Address 3
	    #nByte := #aInput_Byte1[3];
	    "DB_KeyenceCheckerIV3".aDev[#I_nID].In.CommandStatus.bClassificationModeInformation := #nByte.%X0;
	    "DB_KeyenceCheckerIV3".aDev[#I_nID].In.CommandStatus.bReserved5 := #nByte.%X1;
	    "DB_KeyenceCheckerIV3".aDev[#I_nID].In.CommandStatus.bReserved6 := #nByte.%X2;
	    "DB_KeyenceCheckerIV3".aDev[#I_nID].In.CommandStatus.bReserved7 := #nByte.%X3;
	    "DB_KeyenceCheckerIV3".aDev[#I_nID].In.CommandStatus.bSDCardStorageShortage := #nByte.%X4;
	    "DB_KeyenceCheckerIV3".aDev[#I_nID].In.CommandStatus.bBufferOverrun := #nByte.%X5;
	    "DB_KeyenceCheckerIV3".aDev[#I_nID].In.CommandStatus.bWarning := #nByte.%X6;
	    "DB_KeyenceCheckerIV3".aDev[#I_nID].In.CommandStatus.bError := #nByte.%X7;
	    
	    //设备结果/Device Results Bits
	    //Address 0
	    #nByte := #aInput_Byte2[0];
	    "DB_KeyenceCheckerIV3".aDev[#I_nID].In.DeviceResults.bOverallJudgmentOK := #nByte.%X0;
	    "DB_KeyenceCheckerIV3".aDev[#I_nID].In.DeviceResults.bPositionCorrection := #nByte.%X1;
	    "DB_KeyenceCheckerIV3".aDev[#I_nID].In.DeviceResults.bLogic1 := #nByte.%X2;
	    "DB_KeyenceCheckerIV3".aDev[#I_nID].In.DeviceResults.bLogic2 := #nByte.%X3;
	    "DB_KeyenceCheckerIV3".aDev[#I_nID].In.DeviceResults.bLogic3 := #nByte.%X4;
	    "DB_KeyenceCheckerIV3".aDev[#I_nID].In.DeviceResults.bLogic4 := #nByte.%X5;
	    "DB_KeyenceCheckerIV3".aDev[#I_nID].In.DeviceResults.bOverallJudgmentNG := #nByte.%X6;
	    "DB_KeyenceCheckerIV3".aDev[#I_nID].In.DeviceResults.bReserved1 := #nByte.%X7;
	    //Address 1
	    #nByte := #aInput_Byte2[1];
	    "DB_KeyenceCheckerIV3".aDev[#I_nID].In.DeviceResults.nReserved2 := #nByte;
	    //Address 2
	    #nByte := #aInput_Byte2[2];
	    "DB_KeyenceCheckerIV3".aDev[#I_nID].In.DeviceResults.aToolResult[1] := #nByte.%X0;
	    "DB_KeyenceCheckerIV3".aDev[#I_nID].In.DeviceResults.aToolResult[2] := #nByte.%X1;
	    "DB_KeyenceCheckerIV3".aDev[#I_nID].In.DeviceResults.aToolResult[3] := #nByte.%X2;
	    "DB_KeyenceCheckerIV3".aDev[#I_nID].In.DeviceResults.aToolResult[4] := #nByte.%X3;
	    "DB_KeyenceCheckerIV3".aDev[#I_nID].In.DeviceResults.aToolResult[5] := #nByte.%X4;
	    "DB_KeyenceCheckerIV3".aDev[#I_nID].In.DeviceResults.aToolResult[6] := #nByte.%X5;
	    "DB_KeyenceCheckerIV3".aDev[#I_nID].In.DeviceResults.aToolResult[7] := #nByte.%X6;
	    "DB_KeyenceCheckerIV3".aDev[#I_nID].In.DeviceResults.aToolResult[8] := #nByte.%X7;
	    //Address 3
	    #nByte := #aInput_Byte2[3];
	    "DB_KeyenceCheckerIV3".aDev[#I_nID].In.DeviceResults.aToolResult[9] := #nByte.%X0;
	    "DB_KeyenceCheckerIV3".aDev[#I_nID].In.DeviceResults.aToolResult[10] := #nByte.%X1;
	    "DB_KeyenceCheckerIV3".aDev[#I_nID].In.DeviceResults.aToolResult[11] := #nByte.%X2;
	    "DB_KeyenceCheckerIV3".aDev[#I_nID].In.DeviceResults.aToolResult[12] := #nByte.%X3;
	    "DB_KeyenceCheckerIV3".aDev[#I_nID].In.DeviceResults.aToolResult[13] := #nByte.%X4;
	    "DB_KeyenceCheckerIV3".aDev[#I_nID].In.DeviceResults.aToolResult[14] := #nByte.%X5;
	    "DB_KeyenceCheckerIV3".aDev[#I_nID].In.DeviceResults.aToolResult[15] := #nByte.%X6;
	    "DB_KeyenceCheckerIV3".aDev[#I_nID].In.DeviceResults.aToolResult[16] := #nByte.%X7;
	    
	    //设备状态/Device status words
	    //错误编号/Error number
	    #aWord[0] := #aInput_Byte3[0];
	    #aWord[1] := #aInput_Byte3[1];
	    "DB_KeyenceCheckerIV3".aDev[#I_nID].In."DeviceStatus".nErrorNo := #nWord;
	    //警报编号/Warning number
	    #aWord[0] := #aInput_Byte3[2];
	    #aWord[1] := #aInput_Byte3[3];
	    "DB_KeyenceCheckerIV3".aDev[#I_nID].In."DeviceStatus".nWarningNo := #nWord;
	    //剩余缓存数/Number of remaining buffers
	    #aWord[0] := #aInput_Byte3[4];
	    #aWord[1] := #aInput_Byte3[5];
	    "DB_KeyenceCheckerIV3".aDev[#I_nID].In."DeviceStatus".nNumberOfRemainingBuffers := #nWord;
	    //设定校验和/Check sum
	    #aWord[0] := #aInput_Byte3[6];
	    #aWord[1] := #aInput_Byte3[7];
	    "DB_KeyenceCheckerIV3".aDev[#I_nID].In."DeviceStatus".nChecksum := #nWord;
	    //当前程序编号/Current program number
	    #aWord[0] := #aInput_Byte3[8];
	    #aWord[1] := #aInput_Byte3[9];
	    "DB_KeyenceCheckerIV3".aDev[#I_nID].In."DeviceStatus".nCurrentProgramNo := #nWord;
	    //判断时程序编号/Program number during judgment
	    #aWord[0] := #aInput_Byte3[10];
	    #aWord[1] := #aInput_Byte3[11];
	    "DB_KeyenceCheckerIV3".aDev[#I_nID].In."DeviceStatus".nProgramNoDuringJudgment := #nWord;
	    //结果编号/Result number
	    #aWord[0] := #aInput_Byte3[12];
	    #aWord[1] := #aInput_Byte3[13];
	    "DB_KeyenceCheckerIV3".aDev[#I_nID].In."DeviceStatus".nResultNo := #nWord;
	    //处理时间/Processing time
	    #aWord[0] := #aInput_Byte3[14];
	    #aWord[1] := #aInput_Byte3[15];
	    "DB_KeyenceCheckerIV3".aDev[#I_nID].In."DeviceStatus".nProcessingtime := #nWord;
	    
	    //设备统计/Device Statistics
	    //最大处理时间/Processing time max
	    #aWord[0] := #aInput_Byte4[0];
	    #aWord[1] := #aInput_Byte4[1];
	    "DB_KeyenceCheckerIV3".aDev[#I_nID].In."DeviceStatistics".nProcessingTimeMAX := #nWord;
	    //最小处理时间/Processing time min
	    #aWord[0] := #aInput_Byte4[2];
	    #aWord[1] := #aInput_Byte4[3];
	    "DB_KeyenceCheckerIV3".aDev[#I_nID].In."DeviceStatistics".nProcessingTimeMIN := #nWord;
	    //平均处理时间/Processing time average
	    #aWord[0] := #aInput_Byte4[4];
	    #aWord[1] := #aInput_Byte4[5];
	    "DB_KeyenceCheckerIV3".aDev[#I_nID].In."DeviceStatistics".nProcessingTimeAVE := #nWord;
	    //系统预约/Reserved by system
	    #aWord[0] := #aInput_Byte4[6];
	    #aWord[1] := #aInput_Byte4[7];
	    "DB_KeyenceCheckerIV3".aDev[#I_nID].In."DeviceStatistics".nReserved1 := #nWord;
	    //触发次数/Number of triggers
	    #aDWord[0] := #aInput_Byte4[8];
	    #aDWord[1] := #aInput_Byte4[9];
	    #aDWord[2] := #aInput_Byte4[10];
	    #aDWord[3] := #aInput_Byte4[11];
	    "DB_KeyenceCheckerIV3".aDev[#I_nID].In."DeviceStatistics".nNumberOfTriggers := #nDWord;
	    //OK 次数或分类次数/Number of OKs OR Classification number
	    #aDWord[0] := #aInput_Byte4[12];
	    #aDWord[1] := #aInput_Byte4[13];
	    #aDWord[2] := #aInput_Byte4[14];
	    #aDWord[3] := #aInput_Byte4[15];
	    "DB_KeyenceCheckerIV3".aDev[#I_nID].In."DeviceStatistics".nNumberOfOKs := #nDWord;
	    //NG 次数/Number of NGs
	    #aDWord[0] := #aInput_Byte4[16];
	    #aDWord[1] := #aInput_Byte4[17];
	    #aDWord[2] := #aInput_Byte4[18];
	    #aDWord[3] := #aInput_Byte4[19];
	    "DB_KeyenceCheckerIV3".aDev[#I_nID].In."DeviceStatistics".nNumberOfNGs := #nDWord;
	    //触发错误次数/Number of trigger errors
	    #aDWord[0] := #aInput_Byte4[20];
	    #aDWord[1] := #aInput_Byte4[21];
	    #aDWord[2] := #aInput_Byte4[22];
	    #aDWord[3] := #aInput_Byte4[23];
	    "DB_KeyenceCheckerIV3".aDev[#I_nID].In."DeviceStatistics".nNumberOfTriggerErrors := #nDWord;
	    //系统预约/Reserved by system
	    #aDWord[0] := #aInput_Byte4[24];
	    #aDWord[1] := #aInput_Byte4[25];
	    #aDWord[2] := #aInput_Byte4[26];
	    #aDWord[3] := #aInput_Byte4[27];
	    "DB_KeyenceCheckerIV3".aDev[#I_nID].In."DeviceStatistics".nReserved2 := #nDWord;
	    
	    //位置修正结果/Position Adjust Result
	    //位置修正分数/Position correction tool matching rate
	    #aWord[0] := #aInput_Byte5[0];
	    #aWord[1] := #aInput_Byte5[1];
	    "DB_KeyenceCheckerIV3".aDev[#I_nID].In."PositionAdjustResult".nPositionCorrectionToolMatchingRate := #nWord;
	    //最大位置修正分数/Position correction tool matching rate max
	    #aWord[0] := #aInput_Byte5[2];
	    #aWord[1] := #aInput_Byte5[3];
	    "DB_KeyenceCheckerIV3".aDev[#I_nID].In."PositionAdjustResult".nPositionCorrectionToolMatchingRateMAX := #nWord;
	    //最小位置修正分数/Position correction tool matching rate min
	    #aWord[0] := #aInput_Byte5[4];
	    #aWord[1] := #aInput_Byte5[5];
	    "DB_KeyenceCheckerIV3".aDev[#I_nID].In."PositionAdjustResult".nPositionCorrectionToolMatchingRateMIN := #nWord;
	    //位置修正分数下限阈值/Position correction tool threshold
	    #aWord[0] := #aInput_Byte5[6];
	    #aWord[1] := #aInput_Byte5[7];
	    "DB_KeyenceCheckerIV3".aDev[#I_nID].In."PositionAdjustResult".nPositionCorrectionToolThreshold := #nWord;
	    //系统预约/Reserved by system
	    #aWord[0] := #aInput_Byte5[8];
	    #aWord[1] := #aInput_Byte5[9];
	    "DB_KeyenceCheckerIV3".aDev[#I_nID].In."PositionAdjustResult".nReserved1 := #nWord;
	    //系统预约/Reserved by system
	    #aWord[0] := #aInput_Byte5[10];
	    #aWord[1] := #aInput_Byte5[11];
	    "DB_KeyenceCheckerIV3".aDev[#I_nID].In."PositionAdjustResult".nReserved2 := #nWord;
	    //系统预约/Reserved by system
	    #aWord[0] := #aInput_Byte5[12];
	    #aWord[1] := #aInput_Byte5[13];
	    "DB_KeyenceCheckerIV3".aDev[#I_nID].In."PositionAdjustResult".nReserved3 := #nWord;
	    //系统预约/Reserved by system
	    #aWord[0] := #aInput_Byte5[14];
	    #aWord[1] := #aInput_Byte5[15];
	    "DB_KeyenceCheckerIV3".aDev[#I_nID].In."PositionAdjustResult".nReserved4 := #nWord;
	    //系统预约/Reserved by system
	    #aWord[0] := #aInput_Byte5[16];
	    #aWord[1] := #aInput_Byte5[17];
	    "DB_KeyenceCheckerIV3".aDev[#I_nID].In."PositionAdjustResult".nReserved5 := #nWord;
	    //系统预约/Reserved by system
	    #aWord[0] := #aInput_Byte5[18];
	    #aWord[1] := #aInput_Byte5[19];
	    "DB_KeyenceCheckerIV3".aDev[#I_nID].In."PositionAdjustResult".nReserved6 := #nWord;
	    
	    //工具处理结果/Tool Results
	    FOR #nIdx := 1 TO 64 BY 1 DO
	        //工具相似度/Tool matching rate
	        #aWord[0] := #aInput_Byte6[#nIdx - 1].bInput_Byte0;
	        #aWord[1] := #aInput_Byte6[#nIdx - 1].bInput_Byte1;
	        "DB_KeyenceCheckerIV3".aDev[#I_nID].In.ToolResult[#nIdx].nToolMatchingRate := #nWord;
	        //最大工具相似度/Tool matching rate max
	        #aWord[0] := #aInput_Byte6[#nIdx - 1].bInput_Byte2;
	        #aWord[1] := #aInput_Byte6[#nIdx - 1].bInput_Byte3;
	        "DB_KeyenceCheckerIV3".aDev[#I_nID].In.ToolResult[#nIdx].nToolMatchingRateMAX := #nWord;
	        //最小工具相似度/Tool matching rate min
	        #aWord[0] := #aInput_Byte6[#nIdx - 1].bInput_Byte4;
	        #aWord[1] := #aInput_Byte6[#nIdx - 1].bInput_Byte5;
	        "DB_KeyenceCheckerIV3".aDev[#I_nID].In.ToolResult[#nIdx].nToolMatchingRateMIN := #nWord;
	        //工具下限阈值/Tool lower limit value
	        #aWord[0] := #aInput_Byte6[#nIdx - 1].bInput_Byte6;
	        #aWord[1] := #aInput_Byte6[#nIdx - 1].bInput_Byte7;
	        "DB_KeyenceCheckerIV3".aDev[#I_nID].In.ToolResult[#nIdx].nToolLowerLimitValue := #nWord;
	        //工具上限阈值/Tool upper limit value
	        #aWord[0] := #aInput_Byte6[#nIdx - 1].bInput_Byte8;
	        #aWord[1] := #aInput_Byte6[#nIdx - 1].bInput_Byte9;
	        "DB_KeyenceCheckerIV3".aDev[#I_nID].In.ToolResult[#nIdx].nToolUpperLimitValue := #nWord;
	        //小数点位置/Decimal position
	        #aWord[0] := #aInput_Byte6[#nIdx - 1].bInput_Byte10;
	        #aWord[1] := #aInput_Byte6[#nIdx - 1].bInput_Byte11;
	        "DB_KeyenceCheckerIV3".aDev[#I_nID].In.ToolResult[#nIdx].nDecimalPosition := #nWord;
	        //间距当前值 MAX&彩色识别 H（色相）/Pitch present value MAX&color average H (hue)
	        #aWord[0] := #aInput_Byte6[#nIdx - 1].bInput_Byte12;
	        #aWord[1] := #aInput_Byte6[#nIdx - 1].bInput_Byte13;
	        "DB_KeyenceCheckerIV3".aDev[#I_nID].In.ToolResult[#nIdx]."nPitchPresentValueMAX/ColorAverageH (hue)" := #nWord;
	        //间距当前值 MIN&彩色识别 S（彩度）/Pitch present value MIN&color average S
	        #aWord[0] := #aInput_Byte6[#nIdx - 1].bInput_Byte14;
	        #aWord[1] := #aInput_Byte6[#nIdx - 1].bInput_Byte15;
	        "DB_KeyenceCheckerIV3".aDev[#I_nID].In.ToolResult[#nIdx]."nPitchPresentValueMIN/ColorAverageS(saturation)" := #nWord;
	        //间距数量&彩色识别 V（彩度）&亮度平均亮度/Number of pitches&color average V (brightness)&brightness average 
	        #aWord[0] := #aInput_Byte6[#nIdx - 1].bInput_Byte16;
	        #aWord[1] := #aInput_Byte6[#nIdx - 1].bInput_Byte17;
	        "DB_KeyenceCheckerIV3".aDev[#I_nID].In.ToolResult[#nIdx]."nNumberOfPitches/ColorAverageV(brightness)/BrightnessAverage" := #nWord;
	        //系统预约/Reserved by system
	        #aWord[0] := #aInput_Byte6[#nIdx - 1].bInput_Byte18;
	        #aWord[1] := #aInput_Byte6[#nIdx - 1].bInput_Byte19;
	        "DB_KeyenceCheckerIV3".aDev[#I_nID].In.ToolResult[#nIdx].nReserved1 := #nWord;
	    END_FOR;
	    
	    //设备结果/Device Results Bits 
	    //主控编号/The master number
	    #aWord[0] := #aInput_Byte7[0];
	    #aWord[1] := #aInput_Byte7[1];
	    "DB_KeyenceCheckerIV3".aDev[#I_nID].In.ExtendedDeviceResult.nMasterNumber := #nWord;
	    //Address 1
	    #nByte := #aInput_Byte7[2];
	    "DB_KeyenceCheckerIV3".aDev[#I_nID].In.ExtendedDeviceResult.aToolResult[17] := #nByte.%X0;
	    "DB_KeyenceCheckerIV3".aDev[#I_nID].In.ExtendedDeviceResult.aToolResult[18] := #nByte.%X1;
	    "DB_KeyenceCheckerIV3".aDev[#I_nID].In.ExtendedDeviceResult.aToolResult[19] := #nByte.%X2;
	    "DB_KeyenceCheckerIV3".aDev[#I_nID].In.ExtendedDeviceResult.aToolResult[20] := #nByte.%X3;
	    "DB_KeyenceCheckerIV3".aDev[#I_nID].In.ExtendedDeviceResult.aToolResult[21] := #nByte.%X4;
	    "DB_KeyenceCheckerIV3".aDev[#I_nID].In.ExtendedDeviceResult.aToolResult[22] := #nByte.%X5;
	    "DB_KeyenceCheckerIV3".aDev[#I_nID].In.ExtendedDeviceResult.aToolResult[23] := #nByte.%X6;
	    "DB_KeyenceCheckerIV3".aDev[#I_nID].In.ExtendedDeviceResult.aToolResult[24] := #nByte.%X7;
	    //Address 2
	    #nByte := #aInput_Byte7[3];
	    "DB_KeyenceCheckerIV3".aDev[#I_nID].In.ExtendedDeviceResult.aToolResult[25] := #nByte.%X0;
	    "DB_KeyenceCheckerIV3".aDev[#I_nID].In.ExtendedDeviceResult.aToolResult[26] := #nByte.%X1;
	    "DB_KeyenceCheckerIV3".aDev[#I_nID].In.ExtendedDeviceResult.aToolResult[27] := #nByte.%X2;
	    "DB_KeyenceCheckerIV3".aDev[#I_nID].In.ExtendedDeviceResult.aToolResult[28] := #nByte.%X3;
	    "DB_KeyenceCheckerIV3".aDev[#I_nID].In.ExtendedDeviceResult.aToolResult[29] := #nByte.%X4;
	    "DB_KeyenceCheckerIV3".aDev[#I_nID].In.ExtendedDeviceResult.aToolResult[30] := #nByte.%X5;
	    "DB_KeyenceCheckerIV3".aDev[#I_nID].In.ExtendedDeviceResult.aToolResult[31] := #nByte.%X6;
	    "DB_KeyenceCheckerIV3".aDev[#I_nID].In.ExtendedDeviceResult.aToolResult[32] := #nByte.%X7;
	    //Address 3
	    #nByte := #aInput_Byte7[4];
	    "DB_KeyenceCheckerIV3".aDev[#I_nID].In.ExtendedDeviceResult.aToolResult[33] := #nByte.%X0;
	    "DB_KeyenceCheckerIV3".aDev[#I_nID].In.ExtendedDeviceResult.aToolResult[34] := #nByte.%X1;
	    "DB_KeyenceCheckerIV3".aDev[#I_nID].In.ExtendedDeviceResult.aToolResult[35] := #nByte.%X2;
	    "DB_KeyenceCheckerIV3".aDev[#I_nID].In.ExtendedDeviceResult.aToolResult[36] := #nByte.%X3;
	    "DB_KeyenceCheckerIV3".aDev[#I_nID].In.ExtendedDeviceResult.aToolResult[37] := #nByte.%X4;
	    "DB_KeyenceCheckerIV3".aDev[#I_nID].In.ExtendedDeviceResult.aToolResult[38] := #nByte.%X5;
	    "DB_KeyenceCheckerIV3".aDev[#I_nID].In.ExtendedDeviceResult.aToolResult[39] := #nByte.%X6;
	    "DB_KeyenceCheckerIV3".aDev[#I_nID].In.ExtendedDeviceResult.aToolResult[40] := #nByte.%X7;
	    //Address 4
	    #nByte := #aInput_Byte7[5];
	    "DB_KeyenceCheckerIV3".aDev[#I_nID].In.ExtendedDeviceResult.aToolResult[41] := #nByte.%X0;
	    "DB_KeyenceCheckerIV3".aDev[#I_nID].In.ExtendedDeviceResult.aToolResult[42] := #nByte.%X1;
	    "DB_KeyenceCheckerIV3".aDev[#I_nID].In.ExtendedDeviceResult.aToolResult[43] := #nByte.%X2;
	    "DB_KeyenceCheckerIV3".aDev[#I_nID].In.ExtendedDeviceResult.aToolResult[44] := #nByte.%X3;
	    "DB_KeyenceCheckerIV3".aDev[#I_nID].In.ExtendedDeviceResult.aToolResult[45] := #nByte.%X4;
	    "DB_KeyenceCheckerIV3".aDev[#I_nID].In.ExtendedDeviceResult.aToolResult[46] := #nByte.%X5;
	    "DB_KeyenceCheckerIV3".aDev[#I_nID].In.ExtendedDeviceResult.aToolResult[47] := #nByte.%X6;
	    "DB_KeyenceCheckerIV3".aDev[#I_nID].In.ExtendedDeviceResult.aToolResult[48] := #nByte.%X7;
	    //Address 5
	    #nByte := #aInput_Byte7[6];
	    "DB_KeyenceCheckerIV3".aDev[#I_nID].In.ExtendedDeviceResult.aToolResult[49] := #nByte.%X0;
	    "DB_KeyenceCheckerIV3".aDev[#I_nID].In.ExtendedDeviceResult.aToolResult[50] := #nByte.%X1;
	    "DB_KeyenceCheckerIV3".aDev[#I_nID].In.ExtendedDeviceResult.aToolResult[51] := #nByte.%X2;
	    "DB_KeyenceCheckerIV3".aDev[#I_nID].In.ExtendedDeviceResult.aToolResult[52] := #nByte.%X3;
	    "DB_KeyenceCheckerIV3".aDev[#I_nID].In.ExtendedDeviceResult.aToolResult[53] := #nByte.%X4;
	    "DB_KeyenceCheckerIV3".aDev[#I_nID].In.ExtendedDeviceResult.aToolResult[54] := #nByte.%X5;
	    "DB_KeyenceCheckerIV3".aDev[#I_nID].In.ExtendedDeviceResult.aToolResult[55] := #nByte.%X6;
	    "DB_KeyenceCheckerIV3".aDev[#I_nID].In.ExtendedDeviceResult.aToolResult[56] := #nByte.%X7;
	    //Address 6
	    #nByte := #aInput_Byte7[7];
	    "DB_KeyenceCheckerIV3".aDev[#I_nID].In.ExtendedDeviceResult.aToolResult[57] := #nByte.%X0;
	    "DB_KeyenceCheckerIV3".aDev[#I_nID].In.ExtendedDeviceResult.aToolResult[58] := #nByte.%X1;
	    "DB_KeyenceCheckerIV3".aDev[#I_nID].In.ExtendedDeviceResult.aToolResult[59] := #nByte.%X2;
	    "DB_KeyenceCheckerIV3".aDev[#I_nID].In.ExtendedDeviceResult.aToolResult[60] := #nByte.%X3;
	    "DB_KeyenceCheckerIV3".aDev[#I_nID].In.ExtendedDeviceResult.aToolResult[61] := #nByte.%X4;
	    "DB_KeyenceCheckerIV3".aDev[#I_nID].In.ExtendedDeviceResult.aToolResult[62] := #nByte.%X5;
	    "DB_KeyenceCheckerIV3".aDev[#I_nID].In.ExtendedDeviceResult.aToolResult[63] := #nByte.%X6;
	    "DB_KeyenceCheckerIV3".aDev[#I_nID].In.ExtendedDeviceResult.aToolResult[64] := #nByte.%X7;
	END_REGION
	
	REGION CallAdditionalFunctionBlock()
	    //************************************************************************************************
	    //调用外部功能块/Call additional function block
	    //************************************************************************************************
	END_REGION
	
